XV_Alim_Douche(
    Enable := Option_Douche AND NOT Option_Debitmetre_Douche,
    Type_Consigne := FALSE,
    Mode_Vidange := FALSE,
    Cons_Pos_Dem := 0.0,
    Cmd_Ouv_Dem := Cmd_Appli_Vanne_Alim_Douche,
    Info_Mes_Pos := 0.0,
    Presence_Fdc := 3,
    Info_Fdc_Ouvert := E_Vanne_Alim_Douche_Ouv,
    Info_Fdc_Ferme := E_Vanne_Alim_Douche_Ferm,
    Secu_Niveau_Haut := Defaut_Debordement_Douche,
    Defaut_Alim_Eau := Defaut_General_Alim_Eau,
    Control_Discrodance := TRUE,
    Hyst_Al_Discord := 0.0,
    Tempo_Discord_TOR := T#15s,
    EF_Forcage := EF_Cmd_Vanne_Alim_Douche,
    F_STOR_Registre := F_Cmd_Vanne_Alim_Douche,
    F_SAN_Registre := 0.0,
    In_SCL_MIN_REAL := 0.0,
    In_SCL_OUT_REAL := 100.0,
    SAN_MIN := 0.0,
    SAN_MAX := 32767.0); // Registre_V1
S_Cmd_Vanne_Alim_Douche := XV_Alim_Douche.STOR_Cmd_Ouv_Registre;
Defaut_Discord_Vanne_Alim_Douche_Ouv := XV_Alim_Douche.Def_Discordance_Ouverture;
Defaut_Discord_Vanne_Alim_Douche_Ferm := XV_Alim_Douche.Def_Discordance_Fermeture;
XV_Alim_Douchette(
    Enable := Option_Douchette,
    Type_Consigne := FALSE,
    Mode_Vidange := FALSE,
    Cons_Pos_Dem := 0.0,
    Cmd_Ouv_Dem := Cmd_Appli_Vanne_Alim_Douchette,
    Info_Mes_Pos := 0.0,
    Presence_Fdc := 3,
    Info_Fdc_Ouvert := E_Vanne_Alim_Douchette_Ouv,
    Info_Fdc_Ferme := E_Vanne_Alim_Douchette_Ferm,
    Secu_Niveau_Haut := Defaut_Debordement_Douche,
    Defaut_Alim_Eau := Defaut_General_Alim_Eau,
    Control_Discrodance := TRUE,
    Hyst_Al_Discord := 0.0,
    Tempo_Discord_TOR := T#15s,
    EF_Forcage := EF_Cmd_Vanne_Alim_Douchette,
    F_STOR_Registre := F_Cmd_Vanne_Alim_Douchette,
    F_SAN_Registre := 0.0,
    In_SCL_MIN_REAL := 0.0,
    In_SCL_OUT_REAL := 100.0,
    SAN_MIN := 0.0,
    SAN_MAX := 32767.0); // Registre_V1
S_Cmd_Vanne_Alim_Douchette := XV_Alim_Douchette.STOR_Cmd_Ouv_Registre;
Defaut_Discord_Vanne_Alim_Douchette_Ouv := XV_Alim_Douchette.Def_Discordance_Ouverture;
Defaut_Discord_Vanne_Alim_Douchette_Ferm := XV_Alim_Douchette.Def_Discordance_Fermeture;
XV_Alim_Lavabo(
    Enable := Option_Lavabo AND NOT Option_Debitmetre_Lavabo,
    Type_Consigne := FALSE,
    Mode_Vidange := FALSE,
    Cons_Pos_Dem := 0.0,
    Cmd_Ouv_Dem := Cmd_Appli_Vanne_Alim_Lavabo,
    Info_Mes_Pos := 0.0,
    Presence_Fdc := 3,
    Info_Fdc_Ouvert := E_Vanne_Alim_Lavabo_Ouv,
    Info_Fdc_Ferme := E_Vanne_Alim_Lavabo_Ferm,
    Secu_Niveau_Haut := Defaut_Debordement_Lavabo,
    Defaut_Alim_Eau := Defaut_General_Alim_Eau,
    Control_Discrodance := TRUE,
    Hyst_Al_Discord := 0.0,
    Tempo_Discord_TOR := T#15s,
    EF_Forcage := EF_Cmd_Vanne_Alim_Lavabo,
    F_STOR_Registre := F_Cmd_Vanne_Alim_Lavabo,
    F_SAN_Registre := 0.0,
    In_SCL_MIN_REAL := 0.0,
    In_SCL_OUT_REAL := 100.0,
    SAN_MIN := 0.0,
    SAN_MAX := 32767.0); // Registre_V1
S_Cmd_Vanne_Alim_Lavabo := XV_Alim_Lavabo.STOR_Cmd_Ouv_Registre;
Defaut_Discord_Vanne_Alim_Lavabo_Ouv := XV_Alim_Lavabo.Def_Discordance_Ouverture;
Defaut_Discord_Vanne_Alim_Lavabo_Ferm := XV_Alim_Lavabo.Def_Discordance_Fermeture;
XV_Vid_Douche(
    Enable := Option_Douche,
    Type_Consigne := FALSE,
    Mode_Vidange := TRUE,
    Cons_Pos_Dem := 0.0,
    Cmd_Ouv_Dem := Cmd_Appli_Vanne_Vid_Douche OR Mode_Cabine_Libre,
    Info_Mes_Pos := 0.0,
    Presence_Fdc := 3,
    Info_Fdc_Ouvert := E_Vanne_Vidange_Douche_Ouv,
    Info_Fdc_Ferme := E_Vanne_Vidange_Douche_Ferm,
    Secu_Niveau_Haut := Defaut_Debordement_Douche,
    Defaut_Alim_Eau := FALSE,
    Control_Discrodance := TRUE,
    Hyst_Al_Discord := 0.0,
    Tempo_Discord_TOR := T#15s,
    EF_Forcage := EF_Cmd_Vanne_Vid_Douche,
    F_STOR_Registre := F_Cmd_Vanne_Vid_Douche,
    F_SAN_Registre := 0.0,
    In_SCL_MIN_REAL := 0.0,
    In_SCL_OUT_REAL := 100.0,
    SAN_MIN := 0.0,
    SAN_MAX := 32767.0); // Registre_V1
S_Cmd_Vanne_Vid_Douche := XV_Vid_Douche.STOR_Cmd_Ouv_Registre;
Defaut_Discord_Vanne_Vid_Douche_Ouv := XV_Vid_Douche.Def_Discordance_Ouverture;
Defaut_Discord_Vanne_Vid_Douche_Ferm := XV_Vid_Douche.Def_Discordance_Fermeture;
XV_Vid_Lavabo(
    Enable := Option_Lavabo,
    Type_Consigne := FALSE,
    Mode_Vidange := TRUE,
    Cons_Pos_Dem := 0.0,
    Cmd_Ouv_Dem := Cmd_Appli_Vanne_Vid_Lavabo OR Mode_Cabine_Libre,
    Info_Mes_Pos := 0.0,
    Presence_Fdc := 3,
    Info_Fdc_Ouvert := E_Vanne_Vidange_Lavabo_Ouv,
    Info_Fdc_Ferme := E_Vanne_Vidange_Lavabo_Ferm,
    Secu_Niveau_Haut := Defaut_Debordement_Lavabo,
    Defaut_Alim_Eau := FALSE,
    Control_Discrodance := TRUE,
    Hyst_Al_Discord := 0.0,
    Tempo_Discord_TOR := T#15s,
    EF_Forcage := EF_Cmd_Vanne_Vid_Lavabo,
    F_STOR_Registre := F_Cmd_Vanne_Vid_Lavabo,
    F_SAN_Registre := 0.0,
    In_SCL_MIN_REAL := 0.0,
    In_SCL_OUT_REAL := 100.0,
    SAN_MIN := 0.0,
    SAN_MAX := 32767.0); // Registre_V1
S_Cmd_Vanne_Vid_Lavabo := XV_Vid_Lavabo.STOR_Cmd_Ouv_Registre;
Defaut_Discord_Vanne_Vid_Lavabo_Ouv := XV_Vid_Lavabo.Def_Discordance_Ouverture;
Defaut_Discord_Vanne_Vid_Lavabo_Ferm := XV_Vid_Lavabo.Def_Discordance_Fermeture;
XV_Electrovanne_Douche(
    Enable := Option_Debitmetre_Douche,
    Type_Consigne := FALSE,
    Mode_Vidange := FALSE,
    Cons_Pos_Dem := 0.0,
    Cmd_Ouv_Dem := Cmd_Appli_ElectroValve_Alim_Douche,
    Info_Mes_Pos := 0.0,
    Presence_Fdc := 0,
    Info_Fdc_Ouvert := FALSE,
    Info_Fdc_Ferme := FALSE,
    Secu_Niveau_Haut := Defaut_Debordement_Douche,
    Defaut_Alim_Eau := Defaut_General_Alim_Eau,
    Control_Discrodance := TRUE,
    Hyst_Al_Discord := 0.0,
    Tempo_Discord_TOR := T#15s,
    EF_Forcage := EF_Cmd_ElectroValve_Alim_Douche,
    F_STOR_Registre := F_Cmd_ElectroValve_Alim_Douche,
    F_SAN_Registre := 0.0,
    In_SCL_MIN_REAL := 0.0,
    In_SCL_OUT_REAL := 100.0,
    SAN_MIN := 0.0,
    SAN_MAX := 32767.0); // Registre_V1
S_Cmd_ElectroValve_Alim_Douche := XV_Electrovanne_Douche.STOR_Cmd_Ouv_Registre;
XV_Electrovanne_Lavabo(
    Enable := Option_Debitmetre_Lavabo,
    Type_Consigne := FALSE,
    Mode_Vidange := FALSE,
    Cons_Pos_Dem := 0.0,
    Cmd_Ouv_Dem := Cmd_Appli_ElectroValve_Alim_Lavabo,
    Info_Mes_Pos := 0.0,
    Presence_Fdc := 0,
    Info_Fdc_Ouvert := FALSE,
    Info_Fdc_Ferme := FALSE,
    Secu_Niveau_Haut := Defaut_Debordement_Lavabo,
    Defaut_Alim_Eau := Defaut_General_Alim_Eau,
    Control_Discrodance := TRUE,
    Hyst_Al_Discord := 0.0,
    Tempo_Discord_TOR := T#15s,
    EF_Forcage := EF_Cmd_ElectroValve_Alim_Lavabo,
    F_STOR_Registre := F_Cmd_ElectroValve_Alim_Lavabo,
    F_SAN_Registre := 0.0,
    In_SCL_MIN_REAL := 0.0,
    In_SCL_OUT_REAL := 100.0,
    SAN_MIN := 0.0,
    SAN_MAX := 32767.0); // Registre_V1
S_Cmd_ElectroValve_Alim_Lavabo := XV_Electrovanne_Lavabo.STOR_Cmd_Ouv_Registre;
Prise_Cabine(
    Enable := Option_Prise,
    Cmd_Prise := SEL(EF_Cmd_PC_Cab, TRUE, F_Cmd_PC_Cab),
    Cabine_Seche := Option_Cabine_Seche,
    Statut_Ferm_Reg_Douche := TRUE,
    Statut_Ferm_Lavabo := TRUE,
    Statut_Electrovanne_Douche := FALSE,
    Statut_Electrovanne_Lavabo := FALSE,
    Statut_Def_Prise_Porte_Ouverte := Def_Prise_Porte_Ouverte,
    Statut_Def_Discord_Alim_Prise := Def_Discord_Alim_Prise,
    Statut_Defaut_Discord_PC_Cab := Defaut_Discord_PC_Cab); // Prise
S_Cmd_PC_Cab := Prise_Cabine.STOR_Prise;
XV_Vanne_Souf_Bas_Deb(
    Enable := Option_Bas_Debit,
    Type_Consigne := FALSE,
    Mode_Vidange := FALSE,
    Cons_Pos_Dem := 0.0,
    Cmd_Ouv_Dem := Cmd_Appli_Vanne_Souf_Bas_Deb,
    Info_Mes_Pos := 0.0,
    Presence_Fdc := 3,
    Info_Fdc_Ouvert := E_Vanne_Souf_Bas_Deb_Ouv,
    Info_Fdc_Ferme := E_Vanne_Souf_Bas_Deb_Ferm,
    Secu_Niveau_Haut := FALSE,
    Defaut_Alim_Eau := FALSE,
    Control_Discrodance := TRUE,
    Hyst_Al_Discord := 0.0,
    Tempo_Discord_TOR := T#95s,
    EF_Forcage := EF_Vanne_Souf_Bas_Deb,
    F_STOR_Registre := F_Vanne_Souf_Bas_Deb,
    F_SAN_Registre := 0.0,
    In_SCL_MIN_REAL := 0.0,
    In_SCL_OUT_REAL := 100.0,
    SAN_MIN := 0.0,
    SAN_MAX := 32767.0); // Registre_V1
S_Cmd_Vanne_Souf_Bas_Deb := XV_Vanne_Souf_Bas_Deb.STOR_Cmd_Ouv_Registre;
Defaut_Discord_Vanne_Souf_Bas_Deb_Ouv := XV_Vanne_Souf_Bas_Deb.Def_Discordance_Ouverture;
Defaut_Discord_Vanne_Souf_Bas_Deb_Ferm := XV_Vanne_Souf_Bas_Deb.Def_Discordance_Fermeture;
XV_Vanne_Ext_Bas_Deb(
    Enable := Option_Bas_Debit,
    Type_Consigne := FALSE,
    Mode_Vidange := FALSE,
    Cons_Pos_Dem := 0.0,
    Cmd_Ouv_Dem := Cmd_Appli_Vanne_Ext_Bas_Deb,
    Info_Mes_Pos := 0.0,
    Presence_Fdc := 3,
    Info_Fdc_Ouvert := E_Vanne_Ext_Bas_Deb_Ouv,
    Info_Fdc_Ferme := E_Vanne_Ext_Bas_Deb_Ferm,
    Secu_Niveau_Haut := FALSE,
    Defaut_Alim_Eau := FALSE,
    Control_Discrodance := TRUE,
    Hyst_Al_Discord := 0.0,
    Tempo_Discord_TOR := T#95s,
    EF_Forcage := EF_Vanne_Ext_Bas_Deb,
    F_STOR_Registre := F_Vanne_Ext_Bas_Deb,
    F_SAN_Registre := 0.0,
    In_SCL_MIN_REAL := 0.0,
    In_SCL_OUT_REAL := 100.0,
    SAN_MIN := 0.0,
    SAN_MAX := 32767.0); // Registre_V1
S_Cmd_Vanne_Ext_Bas_Deb := XV_Vanne_Ext_Bas_Deb.STOR_Cmd_Ouv_Registre;
Defaut_Discord_Vanne_Ext_Bas_Deb_Ouv := XV_Vanne_Ext_Bas_Deb.Def_Discordance_Ouverture;
Defaut_Discord_Vanne_Ext_Bas_Deb_Ferm := XV_Vanne_Ext_Bas_Deb.Def_Discordance_Fermeture;
Reg_Etanche_Souf(
    Enable := Option_Reg_Etanche_Souf,
    Type_Consigne := FALSE,
    Mode_Vidange := FALSE,
    Cons_Pos_Dem := 0.0,
    Cmd_Ouv_Dem := Cmd_Appli_Reg_Etanche_Souf,
    Info_Mes_Pos := 0.0,
    Presence_Fdc := 0,
    Info_Fdc_Ouvert := FALSE,
    Info_Fdc_Ferme := FALSE,
    Secu_Niveau_Haut := FALSE,
    Defaut_Alim_Eau := FALSE,
    Control_Discrodance := FALSE,
    Hyst_Al_Discord := 0.0,
    Tempo_Discord_TOR := T#40s,
    EF_Forcage := EF_Cmd_Reg_Etanche_Souf,
    F_STOR_Registre := F_Cmd_Reg_Etanche_Souf,
    F_SAN_Registre := 0.0,
    In_SCL_MIN_REAL := 0.0,
    In_SCL_OUT_REAL := 100.0,
    SAN_MIN := 0.0,
    SAN_MAX := 32767.0); // Registre_V1
S_Cmd_Reg_Etanche_Souf := Reg_Etanche_Souf.STOR_Cmd_Ouv_Registre;
XV_Alim_NEP(
    Enable := Option_NEP,
    Type_Consigne := FALSE,
    Mode_Vidange := FALSE,
    Cons_Pos_Dem := 0.0,
    Cmd_Ouv_Dem := Cmd_Appli_Vanne_Alim_NEP,
    Info_Mes_Pos := 0.0,
    Presence_Fdc := 3,
    Info_Fdc_Ouvert := E_Vanne_Alim_NEP_Ouv,
    Info_Fdc_Ferme := E_Vanne_Alim_NEP_Ferm,
    Secu_Niveau_Haut := FALSE,
    Defaut_Alim_Eau := FALSE,
    Control_Discrodance := TRUE,
    Hyst_Al_Discord := 0.0,
    Tempo_Discord_TOR := T#95s,
    EF_Forcage := EF_Vanne_Alim_NEP,
    F_STOR_Registre := F_Vanne_Alim_NEP,
    F_SAN_Registre := 0.0,
    In_SCL_MIN_REAL := 0.0,
    In_SCL_OUT_REAL := 100.0,
    SAN_MIN := 0.0,
    SAN_MAX := 32767.0); // Registre_V1
S_Cmd_Vanne_NEP := XV_Alim_NEP.STOR_Cmd_Ouv_Registre;
Defaut_Discord_Vanne_Alim_NEP_Ouv := XV_Alim_NEP.Def_Discordance_Ouverture;
Defaut_Discord_Vanne_Alim_NEP_Ferm := XV_Alim_NEP.Def_Discordance_Fermeture;
Y_Verin_WC_GV(
    Enable := Option_WC_GV,
    Type_Consigne := FALSE,
    Mode_Vidange := FALSE,
    Cons_Pos_Dem := 0.0,
    Cmd_Ouv_Dem := Cmd_Appli_Verin_WC_GV,
    Info_Mes_Pos := 0.0,
    Presence_Fdc := 0,
    Info_Fdc_Ouvert := FALSE,
    Info_Fdc_Ferme := FALSE,
    Secu_Niveau_Haut := FALSE,
    Defaut_Alim_Eau := FALSE,
    Control_Discrodance := FALSE,
    Hyst_Al_Discord := 0.0,
    Tempo_Discord_TOR := T#95s,
    EF_Forcage := EF_Cmd_Verin_WC_GV,
    F_STOR_Registre := F_Cmd_Verin_WC_GV,
    F_SAN_Registre := 0.0,
    In_SCL_MIN_REAL := 0.0,
    In_SCL_OUT_REAL := 100.0,
    SAN_MIN := 0.0,
    SAN_MAX := 32767.0); // Registre_V1
S_Cmd_Appli_Verin_WC_GV := Y_Verin_WC_GV.STOR_Cmd_Ouv_Registre;
Y_Verin_WC_PV(
    Enable := Option_WC_PV,
    Type_Consigne := FALSE,
    Mode_Vidange := FALSE,
    Cons_Pos_Dem := 0.0,
    Cmd_Ouv_Dem := Cmd_Appli_Verin_WC_PV,
    Info_Mes_Pos := 0.0,
    Presence_Fdc := 0,
    Info_Fdc_Ouvert := FALSE,
    Info_Fdc_Ferme := FALSE,
    Secu_Niveau_Haut := FALSE,
    Defaut_Alim_Eau := FALSE,
    Control_Discrodance := FALSE,
    Hyst_Al_Discord := 0.0,
    Tempo_Discord_TOR := T#95s,
    EF_Forcage := EF_Cmd_Verin_WC_PV,
    F_STOR_Registre := F_Cmd_Verin_WC_PV,
    F_SAN_Registre := 0.0,
    In_SCL_MIN_REAL := 0.0,
    In_SCL_OUT_REAL := 100.0,
    SAN_MIN := 0.0,
    SAN_MAX := 32767.0); // Registre_V1
S_Cmd_Appli_Verin_WC_PV := Y_Verin_WC_PV.STOR_Cmd_Ouv_Registre;
Gestion_EA_WC(
    OUTPUT_1 := Y_Verin_WC_GV.STOR_Cmd_Ouv_Registre,
    OUTPUT_2 := Y_Verin_WC_PV.STOR_Cmd_Ouv_Registre,
    OUTPUT_3 := FALSE,
    OUTPUT_4 := FALSE,
    SWITCH_SEQUENCE := 0); // Sontay_4RM
S_Cons_Module_Sontay := Gestion_EA_WC.OUT_SAN;

END_PROGRAM

// ---- POUs/Block/Autres/Sontay_4RM.TcPOU
FUNCTION_BLOCK Sontay_4RM
VAR_INPUT
	OUTPUT_1 :BOOL;
	OUTPUT_2 :BOOL;
	OUTPUT_3 :BOOL;
	OUTPUT_4 :BOOL;
	SWITCH_SEQUENCE :INT; (*0=Sequenced / 1=Staged / 1=Binary*)
END_VAR
VAR_OUTPUT
	OUT_SAN :INT;
END_VAR
VAR
	Sortie_Calcul_Sequenced :INT;
	SCL_Sequenced: SCL;
END_VAR

(*Bloc de fonction permettant de gérer le module IO-RM4 de sontay*)

(*Version Sequenced*)
IF (SWITCH_SEQUENCE = 0)
	THEN
	IF (OUTPUT_1) (*La valeur doit être comprise entre 2 et 4 VDC*)
		THEN
		Sortie_Calcul_Sequenced := 3;
	END_IF;
	IF (OUTPUT_2) (*La valeur doit être comprise entre 4 et 6 VDC*)
		THEN
		Sortie_Calcul_Sequenced := 5;
	END_IF;
	IF (OUTPUT_3) (*La valeur doit être comprise entre 6 et 8 VDC*)
		THEN
		Sortie_Calcul_Sequenced := 7;
	END_IF;
	IF (OUTPUT_4) (*La valeur doit être comprise entre 8 et 10 VDC*)
		THEN
		Sortie_Calcul_Sequenced := 9;
	END_IF;
	IF (NOT OUTPUT_1 AND NOT OUTPUT_2 AND NOT OUTPUT_3 AND NOT OUTPUT_4)
		THEN
		Sortie_Calcul_Sequenced := 0;
	END_IF;
END_IF;

(*Mise à l'échelle de la valeur*)
SCL_Sequenced(
	IN_INT:= Sortie_Calcul_Sequenced,
	LIM_MIN_IN_REAL:= 0,
	LIM_MAX_IN_REAL:= 10,
	LIM_MIN_OUT_REAL:= 0.0,
	LIM_MAX_OUT_REAL:= 32767.0,
	OUT_INT=> OUT_SAN);

END_FUNCTION_BLOCK

// ---- POUs/s_InterCom_Esclave.TcPOU
PROGRAM s_InterCom_Esclave
VAR
	fbServer						: FB_LocalServer;
	bEnableServer				: BOOL := TRUE;
	fbSocketCloseAll				: FB_SocketCloseAll :=  ( sSrvNetID := '', tTimeout := DEFAULT_ADS_TIMEOUT );
	bCloseAll					: BOOL := TRUE;
	TON_Def_Client: TON;
	TON_Def_Com: TON;
	i :INT;
END_VAR

fbServer(  sLocalHost := Own_Ip_Adress, nLocalPort := 200 );

IF (bCloseAll OR NOT Option_InterCom) THEN (*On PLC reset or program download close all old connections *)
	bCloseAll := FALSE;
	fbSocketCloseAll( bExecute:= TRUE );
ELSE
	fbSocketCloseAll( bExecute:= FALSE );
END_IF

IF (Option_InterCom)
	THEN
	IF NOT fbSocketCloseAll.bBusy THEN
		fbServer( bEnable := bEnableServer );
	END_IF
	(*Gestion du defaut de communication*)
	TON_Def_Client(IN:= (fbServer.nAcceptedClients = 0), PT:= T#10s); (*Si aucun accepté au démarrage de l'automate*)
	TON_Def_Com(IN:= (fbServer.fbRemoteClient[1].fbServerDataExcha.bError OR TON_Def_Client.Q), PT:= T#20s);
	Defaut_Com_Client := TON_Def_Com.Q;
	(*Initilisation des lectures et ecritures en cas de défaut com*)
	IF (Defaut_Com_Client)
		THEN
		FOR i := 0 TO 29 BY 1 DO
		Tab_Com_Send[i] := 0;
		Tab_Com_Receive[i] := 0;
		END_FOR;
	END_IF;
	ELSE
	TON_Def_Client(IN:=FALSE);
	Defaut_Com_Client := FALSE;
	FOR i := 0 TO 29 BY 1 DO
	Tab_Com_Send[i] := 0;
	Tab_Com_Receive[i] := 0;
	END_FOR;
END_IF;

END_PROGRAM

// ---- POUs/Block/Com_Ip/FB_LocalServer.TcPOU
FUNCTION_BLOCK FB_LocalServer
VAR_INPUT
	sLocalHost					: STRING(15);(* own IP address! *)
	nLocalPort					: UDINT := 0;
	bEnable						: BOOL;
END_VAR
VAR_OUTPUT
	bListening					: BOOL;
	hListener 					: T_HSOCKET;
	nAcceptedClients				: UDINT;
	bBusy						: BOOL;
	bError 						: BOOL;
	nErrId						: UDINT;
END_VAR
VAR
	fbListen	 					: FB_SocketListen := ( sSrvNetID := '', tTimeout := DEFAULT_ADS_TIMEOUT );
	fbClose						: FB_SocketClose := ( sSrvNetID := '', tTimeout := DEFAULT_ADS_TIMEOUT );
	fbConnectTON				: TON := ( PT := T#3s );
	eStep						: E_ServerSteps;
	fbRemoteClient				: ARRAY[1..1] OF FB_RemoteClient;
	i							: UDINT;
END_VAR

CASE eStep OF

	SERVER_STATE_IDLE:
		IF bEnable XOR bListening THEN
			bBusy := TRUE;
			bError := FALSE;
			nErrId := 0;
			IF bEnable THEN
				fbConnectTON( IN := FALSE );
				eStep := SERVER_STATE_LISTENER_OPEN_START;
			ELSE
				eStep := SERVER_STATE_REMOTE_CLIENTS_CLOSE;
			END_IF
		ELSIF bListening THEN
			eStep := SERVER_STATE_REMOTE_CLIENTS_COMM;
		END_IF

	SERVER_STATE_LISTENER_OPEN_START:
		fbConnectTON( IN := TRUE, PT := PLCPRJ_RECONNECT_TIME );
		IF fbConnectTON.Q THEN
			fbConnectTON( IN := FALSE );
			fbListen(  bExecute := FALSE  );
			fbListen(	sLocalHost	:= sLocalHost,
					nLocalPort	:= nLocalPort,
					bExecute	:= TRUE );
			eStep := SERVER_STATE_LISTENER_OPEN_WAIT;
		END_IF

	SERVER_STATE_LISTENER_OPEN_WAIT:
		fbListen( bExecute := FALSE );
		IF NOT fbListen.bBusy THEN
			IF NOT fbListen.bError THEN
				bListening 	:= TRUE;
				hListener 	:= fbListen.hListener;
				eStep 		:= SERVER_STATE_IDLE;
				LogMessage( 'LISTENER socket OPENED!', hListener );
			ELSE
				LogError( 'FB_SocketListen',  fbListen.nErrId );
				nErrId := fbListen.nErrId;
				eStep := SERVER_STATE_ERROR;
			END_IF
		END_IF

	SERVER_STATE_REMOTE_CLIENTS_COMM:
		eStep := SERVER_STATE_IDLE;
		nAcceptedClients := 0;

		FOR i:= 1 TO MAX_CLIENT_CONNECTIONS DO
			fbRemoteClient[ i ]( hListener := hListener, bEnable := TRUE );
			IF NOT  fbRemoteClient[ i ].bBusy AND fbRemoteClient[ i ].bError THEN (*FB_SocketAccept returned error!*)
				eStep := SERVER_STATE_REMOTE_CLIENTS_CLOSE;
				EXIT;
			END_IF

			(* count the number of connected remote clients *)
			IF fbRemoteClient[ i ].bAccepted THEN
				nAcceptedClients := nAcceptedClients + 1;
			END_IF

		END_FOR

	SERVER_STATE_REMOTE_CLIENTS_CLOSE:
		nAcceptedClients := 0;
		eStep := SERVER_STATE_LISTENER_CLOSE_START; (* close listener socket too *)
		FOR i:= 1 TO MAX_CLIENT_CONNECTIONS DO
			fbRemoteClient[ i ]( bEnable := FALSE );(* close all remote client (accepted) sockets *)
			(* check if all remote client sockets are closed *)
			IF fbRemoteClient[ i ].bAccepted THEN
				eStep := SERVER_STATE_REMOTE_CLIENTS_CLOSE; (* stay here and close all remote clients first *)
				nAcceptedClients := nAcceptedClients + 1;
			END_IF
		END_FOR

	SERVER_STATE_LISTENER_CLOSE_START:
		fbClose( bExecute := FALSE );
		fbClose(	hSocket	:= hListener,
				bExecute:= TRUE );
		eStep := SERVER_STATE_LISTENER_CLOSE_WAIT;

	SERVER_STATE_LISTENER_CLOSE_WAIT:
		fbClose( bExecute := FALSE );
		IF NOT fbClose.bBusy THEN
			LogMessage( 'LISTENER socket CLOSED!', hListener );
			bListening := FALSE;
			MEMSET( ADR(hListener), 0, SIZEOF(hListener));
			IF fbClose.bError THEN
				LogError( 'FB_SocketClose (listener)',  fbClose.nErrId );
				nErrId := fbClose.nErrId;
				eStep := SERVER_STATE_ERROR;
			ELSE
				bBusy := FALSE;
				bError := FALSE;
				nErrId := 0;
				eStep := SERVER_STATE_IDLE;
			END_IF
		END_IF

	SERVER_STATE_ERROR:
		bError := TRUE;
		IF bListening THEN
			eStep := SERVER_STATE_REMOTE_CLIENTS_CLOSE;
		ELSE
			bBusy := FALSE;
			eStep := SERVER_STATE_IDLE;
		END_IF

END_CASE

END_FUNCTION_BLOCK

// ---- POUs/Block/Com_Ip/FB_RemoteClient.TcPOU
FUNCTION_BLOCK FB_RemoteClient
VAR_INPUT
	hListener				: T_HSOCKET;
	bEnable 				: BOOL;
END_VAR
VAR_OUTPUT
	bAccepted			: BOOL;
	hSocket				: T_HSOCKET;
	bBusy				: BOOL;
	bError 				: BOOL;
	nErrID				: UDINT;
	sFromClient			: T_MaxString;
END_VAR
VAR
	fbAccept 			: FB_SocketAccept := ( sSrvNetID := '', tTimeout := DEFAULT_ADS_TIMEOUT );
	fbClose				: FB_SocketClose := ( sSrvNetID := '', tTimeout := DEFAULT_ADS_TIMEOUT );
	fbServerDataExcha	: FB_ServerDataExcha;
	fbAcceptTON			: TON := ( PT := T#1s);
	eStep				: E_ClientSteps;
	R_TRIG_1: R_TRIG;
END_VAR

CASE eStep OF

	CLIENT_STATE_IDLE:
		IF bEnable XOR bAccepted THEN
			bBusy := TRUE;
			bError := FALSE;
			nErrId := 0;
			sFromClient := '';
			IF bEnable THEN
				fbAcceptTON( IN := FALSE );
				eStep := CLIENT_STATE_CONNECT_START;
			ELSE
				eStep := CLIENT_STATE_CLOSE_START;
			END_IF
		ELSIF bAccepted THEN
			eStep := CLIENT_STATE_DATAEXCHA_START;
		ELSE
			bBusy := FALSE;
		END_IF

	CLIENT_STATE_CONNECT_START:
		fbAcceptTON( IN := TRUE, PT := PLCPRJ_ACCEPT_POLLING_TIME );
		IF fbAcceptTON.Q THEN
			fbAcceptTON( IN := FALSE );
			fbAccept(  bExecute := FALSE  );
			fbAccept(	hListener := hListener,
						bExecute:= TRUE );
			eStep := CLIENT_STATE_CONNECT_WAIT;
		END_IF

	CLIENT_STATE_CONNECT_WAIT:
		fbAccept( bExecute := FALSE );
		IF NOT fbAccept.bBusy THEN
			IF NOT fbAccept.bError THEN
				IF fbAccept.bAccepted THEN
					bAccepted := TRUE;
					hSocket := fbAccept.hSocket;
					LogMessage( 'REMOTE client ACCEPTED!', hSocket );
				END_IF
				eStep := CLIENT_STATE_IDLE;
			ELSE
				LogError( 'FB_SocketAccept',  fbAccept.nErrId );
				nErrId := fbAccept.nErrId;
				eStep := CLIENT_STATE_ERROR;
			END_IF
		END_IF

	CLIENT_STATE_DATAEXCHA_START:
		fbServerDataExcha( bExecute := FALSE );
		fbServerDataExcha( 	hSocket := hSocket,
								bExecute := TRUE );
		eStep := CLIENT_STATE_DATAEXCHA_WAIT;

	CLIENT_STATE_DATAEXCHA_WAIT:
		fbServerDataExcha( bExecute := FALSE, sFromClient=>sFromClient );
		IF NOT fbServerDataExcha.bBusy THEN
			IF NOT fbServerDataExcha.bError THEN
				eStep := CLIENT_STATE_IDLE;
			ELSE
				(* possible errors are logged inside of fbServerDataExcha function block *)
				nErrId := fbServerDataExcha.nErrID;
				eStep := CLIENT_STATE_ERROR;
			END_IF
		END_IF

	CLIENT_STATE_CLOSE_START:
		fbClose( bExecute := FALSE );
		fbClose(	hSocket:= hSocket,
				bExecute:= TRUE );
		eStep := CLIENT_STATE_CLOSE_WAIT;

	CLIENT_STATE_CLOSE_WAIT:
		fbClose( bExecute := FALSE );
		IF NOT fbClose.bBusy THEN
			LogMessage( 'REMOTE client CLOSED!', hSocket );
			bAccepted := FALSE;
			MEMSET( ADR( hSocket ), 0, SIZEOF( hSocket ) );
			IF fbClose.bError THEN
				LogError( 'FB_SocketClose (remote client)', fbClose.nErrId );
				nErrId := fbClose.nErrId;
				eStep := CLIENT_STATE_ERROR;
			ELSE
				bBusy := FALSE;
				bError := FALSE;
				nErrId := 0;
				eStep := CLIENT_STATE_IDLE;
			END_IF
		END_IF

	CLIENT_STATE_ERROR:
		bError := TRUE;
		IF bAccepted THEN
			eStep := CLIENT_STATE_CLOSE_START;
		ELSE
			eStep := CLIENT_STATE_IDLE;
			bBusy := FALSE;
		END_IF
END_CASE

R_TRIG_1(CLK:= fbServerDataExcha.bError);
IF(R_TRIG_1.Q)
	THEN
	eStep := CLIENT_STATE_ERROR;
END_IF;

END_FUNCTION_BLOCK

// ---- POUs/Block/Com_Ip/FB_ServerDataExcha.TcPOU
FUNCTION_BLOCK FB_ServerDataExcha
VAR_INPUT
	hSocket			: T_HSOCKET;
	bExecute		: BOOL;
END_VAR
VAR_OUTPUT
	bBusy			: BOOL;
	bError 			: BOOL;
	nErrID			: UDINT;
	sFromClient		: T_MaxString;
END_VAR
VAR
	fbSocketReceive	: FB_SocketReceive := ( sSrvNetId := '', tTimeout := DEFAULT_ADS_TIMEOUT );
	fbSocketSend	: FB_SocketSend :=  ( sSrvNetId := '', tTimeout := DEFAULT_ADS_TIMEOUT );
	eStep			: E_DataExchaSteps;
	RisingEdge		: R_TRIG;
	fbReceiveTON	: TON;
	fbDisconnectTON 	: TON;
	cbReceived, startPos, endPos, idx	: UDINT;
	cbFrame			: UDINT;
	rxBuffer			: ARRAY[0..1000] OF BYTE;
END_VAR

RisingEdge( CLK := bExecute );
CASE eStep OF

	DATAEXCHA_STATE_IDLE:
		IF RisingEdge.Q THEN
			bBusy 	:= TRUE;
			bError 	:= FALSE;
			nErrId 	:= 0;
			fbDisconnectTON( IN := FALSE, PT := T#0s );(* disable timeout check first *)
			fbReceiveTON( IN := FALSE, PT := T#0s ); (* receive first request immediately *)
			eStep 	:= DATAEXCHA_STATE_RECEIVE_START;
		END_IF

	DATAEXCHA_STATE_RECEIVE_START: (* Receive remote client data *)
		fbReceiveTON(  IN := TRUE );
		IF fbReceiveTON.Q THEN
			fbReceiveTON( IN := FALSE );
			fbSocketReceive( bExecute := FALSE );
			fbSocketReceive( 	hSocket		:= hSocket,
							pDest		:= ADR( Tab_Com_Receive ),			(*ADR( rxBuffer ) + cbReceived,*)
							cbLen		:= SIZEOF( Tab_Com_Receive ),		(*SIZEOF( rxBuffer ) - cbReceived,*)
							bExecute	:= TRUE );
			eStep := DATAEXCHA_STATE_RECEIVE_WAIT;
		END_IF

	DATAEXCHA_STATE_RECEIVE_WAIT:
		fbSocketReceive( bExecute := FALSE );
		IF NOT fbSocketReceive.bBusy THEN
			IF NOT fbSocketReceive.bError THEN

				IF (fbSocketReceive.nRecBytes > 0) THEN(* bytes received *)

					startPos 		:= cbReceived;(* rxBuffer array index of first data byte *)
					endPos  		:= cbReceived + fbSocketReceive.nRecBytes  - 1;(* rxBuffer array index of last data byte *)
					cbReceived 	:= cbReceived + fbSocketReceive.nRecBytes;(* calculate the number of received data bytes *)
					cbFrame		:= 0;(* reset frame length *)

					IF cbReceived < SIZEOF( sFromClient ) THEN(* no overflow *)

						fbReceiveTON( IN := FALSE, PT := T#0s ); (* bytes received => increase the read (polling) speed *)
						fbDisconnectTON( IN := FALSE, PT := PLCPRJ_RECEIVE_TIMEOUT );(* bytes received => disable timeout check *)

						(* search for string end delimiter *)
						FOR idx := startPos TO endPos BY 1 DO
							IF rxBuffer[idx] = 0 THEN(* string end delimiter found *)
								cbFrame := idx + 1;(* calculate the length of the received string (inclusive the end delimiter) *)
								MEMCPY(  ADR( sFromClient ), ADR( rxBuffer ), cbFrame );(* copy the received string to the output variable (inclusive the end delimiter) *)
								MEMMOVE( ADR( rxBuffer ), ADR( rxBuffer[cbFrame] ),  cbReceived - cbFrame  );(* move the reamaining data bytes *)
								cbReceived := cbReceived - cbFrame;(* recalculate the reamaining data byte length *)
								eStep := DATAEXCHA_STATE_SEND_START;
								EXIT;
							END_IF
						END_FOR

					ELSE(* there is no more free read buffer space => the answer string should be terminated *)
						LogError( 'FB_SocketReceive (remote client)',  PLCPRJ_ERROR_RECEIVE_BUFFER_OVERFLOW );
						nErrId := PLCPRJ_ERROR_RECEIVE_BUFFER_OVERFLOW;(* buffer overflow !*)
						eStep := DATAEXCHA_STATE_ERROR;
					END_IF

				ELSE(* no bytes received *)
					fbReceiveTON( IN := FALSE, PT := PLCPRJ_RECEIVE_POLLING_TIME );(* no bytes received => decrease the read (polling) speed *)
					fbDisconnectTON( IN := TRUE, PT := PLCPRJ_RECEIVE_TIMEOUT );(* no bytes received => enable timeout check*)
					IF fbDisconnectTON.Q THEN (* timeout error*)
						fbDisconnectTON( IN := FALSE );
						LogError( 'FB_SocketReceive (remote client)',  PLCPRJ_ERROR_RECEIVE_TIMEOUT );
						nErrID := PLCPRJ_ERROR_RECEIVE_TIMEOUT;
						eStep := DATAEXCHA_STATE_ERROR;
					ELSE(* repeat reading *)
						eStep := DATAEXCHA_STATE_RECEIVE_START; (* repeat reading *)
					END_IF
				END_IF
			ELSE(* receive error *)
				LogError( 'FB_SocketReceive (remote client)',  fbSocketReceive.nErrId );
				nErrId := fbSocketReceive.nErrId;
				eStep := DATAEXCHA_STATE_ERROR;
			END_IF
		END_IF

	DATAEXCHA_STATE_SEND_START:
		fbSocketSend( bExecute := FALSE );
		fbSocketSend(	hSocket	:= hSocket,
						pSrc	:= ADR( Tab_Com_Send ),			(*ADR( sFromClient ),*)
						cbLen	:= SIZEOF( Tab_Com_Send ),		(*INT_TO_UDINT(LEN( sFromClient )) + 1,(* string length inclusive the zero delimiter *)*)
						bExecute:= TRUE );
		eStep := DATAEXCHA_STATE_SEND_WAIT;

	DATAEXCHA_STATE_SEND_WAIT:
		fbSocketSend( bExecute := FALSE );
		IF NOT fbSocketSend.bBusy THEN
			IF NOT fbSocketSend.bError THEN
				bBusy := FALSE;
				eStep := DATAEXCHA_STATE_IDLE;
			ELSE
				LogError( 'fbSocketSend (remote client)',  fbSocketSend.nErrId );
				nErrId := fbSocketSend.nErrId;
				eStep := DATAEXCHA_STATE_ERROR;
			END_IF
		END_IF

	DATAEXCHA_STATE_ERROR:
		bBusy := FALSE;
		bError := TRUE;
		cbReceived := 0;(* reset old received data bytes *)
		eStep := DATAEXCHA_STATE_IDLE;
END_CASE

END_FUNCTION_BLOCK

// ---- POUs/Block/Com_Ip/LogError.TcPOU
FUNCTION LogError : DINT
VAR_INPUT
	msg			: STRING;
	nErrId		: DWORD;
END_VAR
VAR
END_VAR

IF bLogDebugMessages THEN
	IF nErrId = 0 THEN
		LogError := ADSLOGSTR( ADSLOG_MSGTYPE_HINT OR ADSLOG_MSGTYPE_LOG, CONCAT( msg, '::No error!   %s'),'' );
	ELSIF ( nErrId AND 16#80000000) =16#80000000 THEN
		LogError := ADSLOGDINT( ADSLOG_MSGTYPE_ERROR OR ADSLOG_MSGTYPE_LOG, CONCAT( msg, ':: Win32 error: %d' ), DWORD_TO_DINT(SCODE_CODE( nErrId )) );
	ELSIF (nErrId AND 16#00008100) =16#00008100 THEN
		LogError := ADSLOGDINT( ADSLOG_MSGTYPE_ERROR OR ADSLOG_MSGTYPE_LOG, CONCAT( msg, '::Internal PLC sample project error: %d' ), DWORD_TO_DINT(nErrId) );
	ELSIF (nErrId AND 16#00008000) =16#00008000 THEN
		LogError := ADSLOGDINT( ADSLOG_MSGTYPE_ERROR OR ADSLOG_MSGTYPE_LOG, CONCAT( msg, '::Internal TCP/IP Connection Server error: %d' ), DWORD_TO_DINT(nErrId) );
	ELSE
		LogError := ADSLOGDINT( ADSLOG_MSGTYPE_ERROR OR ADSLOG_MSGTYPE_LOG, CONCAT( msg, '::TwinCAT System error: %d' ), DWORD_TO_DINT(nErrId) );
	END_IF
END_IF

END_FUNCTION

// ---- POUs/Block/Com_Ip/SCODE_CODE.TcPOU
FUNCTION SCODE_CODE : DWORD
VAR_INPUT
	sc		: DWORD;
END_VAR

SCODE_CODE := 16#FFFF AND sc;

END_FUNCTION

// ---- POUs/Block/Com_Ip/LogMessage.TcPOU
FUNCTION LogMessage : DINT
VAR_INPUT
	msg		: STRING;
	hSocket	: T_HSOCKET;
END_VAR
VAR
END_VAR

IF bLogDebugMessages THEN
	LogMessage := ADSLOGDINT( ADSLOG_MSGTYPE_HINT OR ADSLOG_MSGTYPE_LOG, CONCAT( msg, '::Internal handle: %d' ), UDINT_TO_DINT(hSocket.handle)  );
END_IF

END_FUNCTION

// ---- POUs/t_Enr_Variables.TcPOU
PROGRAM t_Enr_Variables
VAR
	WritePersistentData_1: WritePersistentData;
 	 bStart                : BOOL := TRUE;
  	 bError                : BOOL;
   	 bBusy                 : BOOL;
   	 nErrorId              : UDINT;
	Enregistrement_Manu: BOOL;
	TP_RAZ_Enr_Manu :TP;
END_VAR

TP_RAZ_Enr_Manu(IN:= Enregistrement_Manu, PT:= T#2S);
Enregistrement_Manu := (SEL(Enregistrement_Manu, Enregistrement_Manu, FALSE) OR TP_RAZ_Enr_Manu.Q);

(******************Gestion enregistrement des varaibles perssitantes********************************)
WritePersistentData_1(
	NETID:= '',
	PORT:= 851,
	START:= Enregistrement_Manu OR bStart,
	TMOUT:= T#1s,
	BUSY=> bBusy,
	ERR=> bError,
	ERRID=>nErrorId);
bStart := FALSE;

END_PROGRAM

// ---- POUs/Visualisation/Visu.TcPOU
PROGRAM Visu
VAR
	Info_PLC: FB_GetLocalAmsNetId;
	Start: BOOL;
	//Clignotement pour gérer des animations :
	Tmr         	: TON;   	// temporisateur On-Delay standard
    RTrig       	: R_TRIG;	// détecteur de front montant
	Tmr1         	: TON;   	// temporisateur On-Delay standard
    RTrig1       	: R_TRIG;	// détecteur de front montant
	Tmr2         	: TON;   	// temporisateur On-Delay standard
    RTrig2       	: R_TRIG;	// détecteur de front montant
	Var_Test1		: WSTRING(511);
	Var_Test2		: WSTRING;
	Var_test3		: TIME;
	Var_test4		: BOOL;
	// Gestion de l'affichage de la couleur de la cabine :	
    Opacite 		: BYTE := 66; // Opacité (0 = transparent, 255 = opaque)
	Opacite1 		: BYTE := 150; // Opacité (0 = transparent, 255 = opaque)
	//Gestion du pop-up actionneurs
	On_Off_Ventilation	:BOOL;
	//Gestion de la page Nettoyage
	Cpt_Clean		:INT;
	R_TRIG_Inc: R_TRIG;
	//Gestion de la page Recet_EnCours	
	R_TRIG_RecetEnCours: R_TRIG;
	RS_VolEau_Douche: RS;
	RS_VolEau_Lavabo: RS;
	//Gestion de la page Mode_Manu	
	R_TRIG_RecetEnCours_Manu: R_TRIG;
	RS_VolEau_Douche_Manu: RS;
	RS_VolEau_Lavabo_Manu: RS;
	Manu_Tot_Second:DINT;
	Heure_Limite_Douche:REAL;
	Minute_Limite_Douche:REAL;
	Seconde_Limite_Douche:REAL;
	Heure_Limite_Lavabo:REAL;
	Minute_Limite_Lavabo:REAL;
	Seconde_Limite_Lavabo:REAL;
	Heure_Limite_WC:REAL;
	Minute_Limite_WC:REAL;
	Seconde_Limite_WC:REAL;
	//Gestion de la page menu
	R_Trig_Init: R_TRIG;
	TON_Menu: TON;
	R_TRIG_Menu: R_TRIG;
	//Gestion des pages de pop up des alarmes avec réarmement
	NivHaut :BOOL;
	Alarms	:BOOL;
	F_TRIG_Deco: F_TRIG;
	IHM_Mesure_Debit_Deconta: REAL;
END_VAR

GVL_Visu.Page_En_Cours 	:= VisuElems.CURRENTVISU; 			// Récupération du nom de la page en cours
Var_Test1 				:= VisuElems.CurrentFullUserName;
GVL_Visu.Language 		:= VisuElems.CURRENTLANGUAGE;		// récupération du language en cours
GVL_Visu.Connexion 		:= VisuElems.CurrentUserGroupName;	// Récupération du nom de l'utilisateur en cours (Peu poser problème si plusieurs connexion en même temps)
Var_Test2 				:= VisuElems.CurrentUserName;
Var_test3 				:= VisuElems.CurrentRemainingAutoLogoutTime;
Var_test4 				:= VisuElems.CurrentUseAutoLogoutTime;
Info_PLC(bExecute:= Start, tTimeOut:= DEFAULT_ADS_TIMEOUT);

//////////////////////////////////////////////////////////////
//Gestion de la page dépollution							//
//////////////////////////////////////////////////////////////
// Mouvement de la flèche vers le haut :
IF (Mode_Cabine_Depollution)
	THEN
		GVL_Visu.Arrow_Up := GVL_Visu.Arrow_Up - 1;
		IF (GVL_Visu.Arrow_Up = 0)
			THEN
			GVL_Visu.Arrow_Up := 150;
		END_IF;
	ELSE
		GVL_Visu.Arrow_Up := 150;
END_IF
// Mouvement de la flèche vers le bas :
IF (Mode_Cabine_Depollution)
	THEN
		GVL_Visu.Arrow_Down := LIMIT(0, GVL_Visu.Arrow_Down + 1, 150);
		IF (GVL_Visu.Arrow_Down = 150)
			THEN
			GVL_Visu.Arrow_Down := 0;
		END_IF;
	ELSE
		GVL_Visu.Arrow_Down := 0;
END_IF

// Retour à la page Menu à la fin du mode Depollution
IF ((GVL_Visu.Page_En_Cours = 'Depollution') AND R_TRIG_RecetEnCours_Manu.Q)
	THEN
	VisuElems.CURRENTVISU := 'menu';
END_IF

//Affichage de la valeur de mesure
IHM_Mesure_Debit_Deconta := GVL_RegTROX.MES_RegSouf_GD_FCVT01.Mesure_EAN / LIMIT(1.0, Volume_Cabine, 1000);

//////////////////////////////////////////////////////////////
//Gestion du pop-up actionneurs								//
//////////////////////////////////////////////////////////////
IF (MES_Debit_Volh_Soufflage > 1.0)
	THEN
		On_Off_Ventilation := TRUE;
	ELSE
		On_Off_Ventilation := FALSE;
END_IF

//////////////////////////////////////////////////////////////
//Gestion de la page Nettoyage								//
//////////////////////////////////////////////////////////////
R_TRIG_Inc(CLK:= GVL_Visu.On_Off_Anim_Rap);
IF (R_TRIG_Inc.Q AND Mode_Cabine_Nettoyage)
	THEN
		Cpt_Clean := Cpt_Clean + 1;
		IF (Cpt_Clean > 7)
			THEN
				Cpt_Clean := 0;
		END_IF
END_IF
IF (NOT Mode_Cabine_Nettoyage)
	THEN
		Cpt_Clean := 0;
END_IF
CASE Cpt_Clean OF
	0:	// Etape 0 initialisation des valeurs
	GVL_Visu.Cmd_Img_Clean1 := FALSE;
	GVL_Visu.Cmd_Img_Clean2 := FALSE;
	GVL_Visu.Cmd_Img_Clean3 := FALSE;
	GVL_Visu.Cmd_Img_Clean4 := FALSE;
	GVL_Visu.Cmd_Img_Clean5 := FALSE;
	GVL_Visu.Cmd_Img_Clean6 := FALSE;
	GVL_Visu.Cmd_Img_Clean7 := FALSE;
	
	1: // Etape affichage de l'image 1
	GVL_Visu.Cmd_Img_Clean1 := TRUE;
	GVL_Visu.Cmd_Img_Clean2 := FALSE;
	GVL_Visu.Cmd_Img_Clean3 := FALSE;
	GVL_Visu.Cmd_Img_Clean4 := FALSE;
	GVL_Visu.Cmd_Img_Clean5 := FALSE;
	GVL_Visu.Cmd_Img_Clean6 := FALSE;
	GVL_Visu.Cmd_Img_Clean7 := FALSE;
	
	2: // Etape affichage de l'image 1,2
	GVL_Visu.Cmd_Img_Clean1 := TRUE;
	GVL_Visu.Cmd_Img_Clean2 := TRUE;
	GVL_Visu.Cmd_Img_Clean3 := FALSE;
	GVL_Visu.Cmd_Img_Clean4 := FALSE;
	GVL_Visu.Cmd_Img_Clean5 := FALSE;
	GVL_Visu.Cmd_Img_Clean6 := FALSE;
	GVL_Visu.Cmd_Img_Clean7 := FALSE;
	
	3: // Etape affichage de l'image 1,2,3
	GVL_Visu.Cmd_Img_Clean1 := TRUE;
	GVL_Visu.Cmd_Img_Clean2 := TRUE;
	GVL_Visu.Cmd_Img_Clean3 := TRUE;
	GVL_Visu.Cmd_Img_Clean4 := FALSE;
	GVL_Visu.Cmd_Img_Clean5 := FALSE;
	GVL_Visu.Cmd_Img_Clean6 := FALSE;
	GVL_Visu.Cmd_Img_Clean7 := FALSE;
	
	4: // Etape affichage de l'image 1,2,3,4
	GVL_Visu.Cmd_Img_Clean1 := TRUE;
	GVL_Visu.Cmd_Img_Clean2 := TRUE;
	GVL_Visu.Cmd_Img_Clean3 := TRUE;
	GVL_Visu.Cmd_Img_Clean4 := TRUE;
	GVL_Visu.Cmd_Img_Clean5 := FALSE;
	GVL_Visu.Cmd_Img_Clean6 := FALSE;
	GVL_Visu.Cmd_Img_Clean7 := FALSE;
	
	5: // Etape affichage de l'image 1,2,3,4,5
	GVL_Visu.Cmd_Img_Clean1 := TRUE;
	GVL_Visu.Cmd_Img_Clean2 := TRUE;
	GVL_Visu.Cmd_Img_Clean3 := TRUE;
	GVL_Visu.Cmd_Img_Clean4 := TRUE;
	GVL_Visu.Cmd_Img_Clean5 := TRUE;
	GVL_Visu.Cmd_Img_Clean6 := FALSE;
	GVL_Visu.Cmd_Img_Clean7 := FALSE;
	
	6: // Etape affichage de l'image 1,2,3,4,5,6
	GVL_Visu.Cmd_Img_Clean1 := TRUE;
	GVL_Visu.Cmd_Img_Clean2 := TRUE;
	GVL_Visu.Cmd_Img_Clean3 := TRUE;
	GVL_Visu.Cmd_Img_Clean4 := TRUE;
	GVL_Visu.Cmd_Img_Clean5 := TRUE;
	GVL_Visu.Cmd_Img_Clean6 := TRUE;
	GVL_Visu.Cmd_Img_Clean7 := FALSE;
	
	7: // Etape affichage de l'image 1,2,3,4,5,6,7
	GVL_Visu.Cmd_Img_Clean1 := TRUE;
	GVL_Visu.Cmd_Img_Clean2 := TRUE;
	GVL_Visu.Cmd_Img_Clean3 := TRUE;
	GVL_Visu.Cmd_Img_Clean4 := TRUE;
	GVL_Visu.Cmd_Img_Clean5 := TRUE;
	GVL_Visu.Cmd_Img_Clean6 := TRUE;
	GVL_Visu.Cmd_Img_Clean7 := TRUE;
END_CASE

// Retour à la page Menu à la fin du mode Nettoyage
IF ((GVL_Visu.Page_En_Cours = 'Nettoyage') AND R_TRIG_RecetEnCours_Manu.Q)
	THEN
	VisuElems.CURRENTVISU := 'menu';
END_IF

//////////////////////////////////////////////////////////////
//Gestion de la page Sel_Recettes							//
//////////////////////////////////////////////////////////////
IF (Nbre_Etape_Totale <> 0)
	THEN
	GVL_Visu.Visu_Btn_Start := FALSE;
	ELSE
	GVL_Visu.Visu_Btn_Start := TRUE;
END_IF

//////////////////////////////////////////////////////////////
//Gestion de la page Recet_EnCours							//
//////////////////////////////////////////////////////////////
//Affichage de la valeur du volume d'eau restant pour la douche - reset de l'affichage quand la vidange est ouverte
RS_VolEau_Douche (SET:= Mode_Auto.Mode_12 OR Mode_Auto.Mode_13, RESET1:= E_Vanne_Vidange_Douche_Ouv OR Mode_Cabine_Libre);
GVL_Visu.Visu_VolEau_Douche := Mode_Auto.Mode_12 OR Mode_Auto.Mode_13;

//Affichage de la valeur du volume d'eau restant pour le lavabo - reset de l'affichage quand la vidange est ouverte
RS_VolEau_Lavabo (SET:= Mode_Auto.Mode_14 OR Mode_Auto.Mode_15, RESET1:= E_Vanne_Vidange_Lavabo_Ouv OR Mode_Cabine_Libre);
GVL_Visu.Visu_VolEau_Lavabo := Mode_Auto.Mode_14 OR Mode_Auto.Mode_15;

//Affichage du décomptes en secondes
GVL_Visu.Visu_Tempo := Mode_Auto.Mode_1 OR Mode_Auto.Mode_2 OR Mode_Auto.Mode_4 OR Mode_Auto.Mode_5 OR Mode_Auto.Mode_6
						OR Mode_Auto.Mode_7 OR Mode_Auto.Mode_8 OR Mode_Auto.Mode_10 OR Mode_Auto.Mode_11
						OR Mode_Auto.Mode_18 OR Mode_Auto.Mode_19 OR Mode_Auto.Mode_27;

//Affichage du nombre de cycle restant de chasse d'eau
GVL_Visu.Visu_ChasseEau := Mode_Auto.Mode_9 OR Mode_Auto.Mode_26;

//Affichage du débit d'eau, peu importe si c'est la douche ou le lavabo
GVL_Visu.Visu_Debit_Eau := Mode_Auto.Mode_14 OR Mode_Auto.Mode_15 OR Mode_Auto.Mode_12 OR Mode_Auto.Mode_13;
GVL_Visu.Visu_Mes_Debit_Eau := MAX(Tab_MES_Sonde_Debit_Alim_Douche.R_MesCor,Tab_MES_Sonde_Debit_Alim_Lavabo.R_MesCor);

// Retour à la page Menu à la fin de la recette
R_TRIG_RecetEnCours(CLK:= Mode_Cabine_Libre);
IF ((GVL_Visu.Page_En_Cours = 'Recet_EnCours') AND R_TRIG_RecetEnCours.Q)
	THEN
	VisuElems.CURRENTVISU := 'menu';
END_IF

//////////////////////////////////////////////////////////////
//Gestion de la page Mode_Manu								//
//////////////////////////////////////////////////////////////
//Affichage de la valeur du volume d'eau restant pour la douche - reset de l'affichage quand la vidange est ouverte
RS_VolEau_Douche_Manu (SET:= Mode_Manu.Mode_12 OR Mode_Manu.Mode_13, RESET1:= Mode_Cabine_Libre);
GVL_Visu.Visu_VolEau_Douche_Manu := RS_VolEau_Douche_Manu.Q1;

//Affichage de la valeur du volume d'eau restant pour le lavabo - reset de l'affichage quand la vidange est ouverte
RS_VolEau_Lavabo_Manu (SET:= Mode_Manu.Mode_14 OR Mode_Manu.Mode_15, RESET1:= Mode_Cabine_Libre);
GVL_Visu.Visu_VolEau_Lavabo_Manu := RS_VolEau_Lavabo_Manu.Q1;

//Affichage du nombre de cycle restant de chasse d'eau
GVL_Visu.Visu_ChasseEau_Manu := Mode_Manu.Mode_9 OR Mode_Manu.Mode_26;

//Affichage du débit d'eau, peu importe si c'est la douche ou le lavabo
GVL_Visu.Visu_Debit_Eau_Manu := Mode_Manu.Mode_14 OR Mode_Manu.Mode_15 OR Mode_Manu.Mode_12 OR Mode_Manu.Mode_13;
GVL_Visu.Visu_Mes_Debit_Eau_Manu := MAX(Tab_MES_Sonde_Debit_Alim_Douche.R_MesCor,Tab_MES_Sonde_Debit_Alim_Lavabo.R_MesCor);

// Retour à la page Menu à la fin du mode manu
R_TRIG_RecetEnCours_Manu(CLK:= Mode_Cabine_Libre);
IF ((GVL_Visu.Page_En_Cours = 'ModeManuel') AND R_TRIG_RecetEnCours_Manu.Q)
	THEN
	VisuElems.CURRENTVISU := 'menu';
END_IF

// Conversion en integer de la variable de sélection du mode
GVL_Visu.Manu_Choix_Numero_Mode_INT := REAL_TO_INT(Manu_Choix_Numero_Mode);

// Gestion de la sélection des modes manuel présent dans le projet :
GVL_Visu.Tab_Choix_Modes[1] := FALSE;		// Mode 1 douche avec vidange avec tempo
GVL_Visu.Tab_Choix_Modes[2] := FALSE;		// Mode 2 douche sans vidange  avec tempo
GVL_Visu.Tab_Choix_Modes[3] := FALSE;		// Mode 3 douchette avec vidange
GVL_Visu.Tab_Choix_Modes[4] := TRUE;		// Mode 4 lavabo avec vidange avec tempo
GVL_Visu.Tab_Choix_Modes[5] := TRUE;		// Mode 5 lavabo sans vidange avec tempo
GVL_Visu.Tab_Choix_Modes[6] := FALSE;		// Mode 6 activation prise
GVL_Visu.Tab_Choix_Modes[7] := TRUE;		// Mode 7 vidange(s)
GVL_Visu.Tab_Choix_Modes[8] := TRUE;		// Mode 8 neutre
GVL_Visu.Tab_Choix_Modes[9] := FALSE;		// Mode 9 CHASSE D EAU GRAND VOLUME
GVL_Visu.Tab_Choix_Modes[10] := FALSE;		// Mode 10 Dépollution
GVL_Visu.Tab_Choix_Modes[11] := FALSE;		// Mode 11 bas débit
GVL_Visu.Tab_Choix_Modes[12] := FALSE;		// Mode 12 douche avec vidange transition volume d'eau
GVL_Visu.Tab_Choix_Modes[13] := FALSE;		// Mode 13 douche sans vidange transition volume d'eau
GVL_Visu.Tab_Choix_Modes[14] := TRUE;		// Mode 14 lavabo avec vidange transition volume d'eau
GVL_Visu.Tab_Choix_Modes[15] := TRUE;		// Mode 15 lavabo sans vidange transition volume d'eau
GVL_Visu.Tab_Choix_Modes[16] := FALSE;		// Mode 16 douche avec vidange avec BP
GVL_Visu.Tab_Choix_Modes[17] := FALSE;		// Mode 17 lavabo avec vidange avec BP
GVL_Visu.Tab_Choix_Modes[18] := FALSE;		// Mode 18 lavage NEP eau chaude
GVL_Visu.Tab_Choix_Modes[19] := FALSE;		// Mode 19 lavage NEP eau froide
GVL_Visu.Tab_Choix_Modes[20] := FALSE;		// Mode 20 Paramétrable (non utilisé)
GVL_Visu.Tab_Choix_Modes[21] := FALSE;		// Mode 21 alerte préparateur
GVL_Visu.Tab_Choix_Modes[22] := FALSE;		// Mode 22 alerte évaluateur
GVL_Visu.Tab_Choix_Modes[23] := FALSE;		// Mode 23 évaluation (sans moteur bypass)
GVL_Visu.Tab_Choix_Modes[24] := FALSE;		// Mode 24 évaluation (avec moteur bypass)
GVL_Visu.Tab_Choix_Modes[25] := FALSE;		// Mode 25 MISE EN CONDITION
GVL_Visu.Tab_Choix_Modes[26] := FALSE;		// Mode 26 CHASSE D EAU PETIT VOLUME
GVL_Visu.Tab_Choix_Modes[27] := FALSE;		// Mode nettoyage (version NEP)
GVL_Visu.Tab_Choix_Modes[28] := FALSE;		// Mode cabine en condition
GVL_Visu.Tab_Choix_Modes[29] := FALSE;		// Libre
GVL_Visu.Tab_Choix_Modes[30] := FALSE;		// Mode 30 à 59 texte éditable
//premier mode
GVL_Visu.Min_Mode_Manu := 4;
//dernier mode
GVL_Visu.Max_Mode_Manu := 15;

//Affichage du paramétrage du débit d'eau Lavabo
GVL_Visu.Affich_Debit_Eau_Manu := (Manu_Choix_Numero_Mode = 14) OR (Manu_Choix_Numero_Mode = 15)
											OR (Manu_Choix_Numero_Mode = 12) OR (Manu_Choix_Numero_Mode = 13);
//Affichage du paramétrage du débit d'eau douche
GVL_Visu.Affich_Debit_Eau_Manu_Douche := (Manu_Choix_Numero_Mode = 12) OR (Manu_Choix_Numero_Mode = 13);
//Affichage du paramétrage du débit d'eau Lavabo
GVL_Visu.Affich_Debit_Eau_Manu_Lavabo := (Manu_Choix_Numero_Mode = 14) OR (Manu_Choix_Numero_Mode = 15);

//Affichage de la consigne de température
GVL_Visu.Visu_Temp_Manu := 	Option_Regul_Temp_Eau AND
							((Manu_Choix_Numero_Mode = 1) OR (Manu_Choix_Numero_Mode = 2)
							OR (Manu_Choix_Numero_Mode = 4) OR (Manu_Choix_Numero_Mode = 5)
							OR (Manu_Choix_Numero_Mode = 12) OR (Manu_Choix_Numero_Mode = 13)
							OR (Manu_Choix_Numero_Mode = 14) OR (Manu_Choix_Numero_Mode = 15));								
									
//Affichage du paramétrage de la chasse d'eau
GVL_Visu.Affich_ChasseEau_Manu := (Manu_Choix_Numero_Mode = 9) OR (Manu_Choix_Numero_Mode = 26);

//Gestion des limites minimum et maximum du volume d'eau lors d'une vidange fermée
IF (Manu_Choix_Numero_Mode = 13)		//Douche
	THEN
	Manu_Lct_Cons_Vol_Douche := LIMIT(0, Manu_Lct_Cons_Vol_Douche, Volume_Secu_Debord_Douche);
	ELSE
	Manu_Lct_Cons_Vol_Douche := LIMIT(0, Manu_Lct_Cons_Vol_Douche, 999);
END_IF
IF (Manu_Choix_Numero_Mode = 15)		//Lavabo
	THEN
	Manu_Lct_Cons_Vol_Lavabo := LIMIT(0, Manu_Lct_Cons_Vol_Lavabo, Volume_Secu_Debord_Lavabo);
	ELSE
	Manu_Lct_Cons_Vol_Lavabo := LIMIT(0, Manu_Lct_Cons_Vol_Lavabo, 999);
END_IF

//Gestion des limites de temporisation lors d'une vidange fermée et du temps de remplissage du WC
Manu_Tot_Second := (TO_DINT(Manu_Tempo_Transition_Heure) * 3600)
					+ (TO_DINT(Manu_Tempo_Transition_Minute) * 60)
					+ (TO_DINT(Manu_Tempo_Transition_Seconde));
//Limite de la sécurité haute de la douche
Seconde_Limite_Douche 	:= TO_REAL((Temp_Secu_Debord_Douche) MOD 60);
Minute_Limite_Douche 	:= TO_REAL((Temp_Secu_Debord_Douche / 60) MOD 60);
Heure_Limite_Douche 	:= TO_REAL((Temp_Secu_Debord_Douche / 3600) MOD 24);
//Limite de la sécurité haute du lavabo
Seconde_Limite_Lavabo	:= TO_REAL((Temp_Secu_Debord_Lavabo) MOD 60);
Minute_Limite_Lavabo 	:= TO_REAL((Temp_Secu_Debord_Lavabo / 60) MOD 60);
Heure_Limite_Lavabo 	:= TO_REAL((Temp_Secu_Debord_Lavabo / 3600) MOD 24);
//Limite de la sécurité haute du cycle de chasse d'eau
Seconde_Limite_WC		:= TO_REAL((Temps_Remplissage_WC) MOD 60);
Minute_Limite_WC 		:= TO_REAL((Temps_Remplissage_WC / 60) MOD 60);
Heure_Limite_WC 		:= TO_REAL((Temps_Remplissage_WC / 3600) MOD 24);
IF (Manu_Choix_Numero_Mode = 2 AND Option_Douche)
	THEN	//Douche
	IF (Manu_Tot_Second > TO_DINT(Temp_Secu_Debord_Douche))
		THEN
		Manu_Tempo_Transition_Seconde := Seconde_Limite_Douche;
		Manu_Tempo_Transition_Minute := Minute_Limite_Douche;
		Manu_Tempo_Transition_Heure := Heure_Limite_Douche;
	END_IF
	ELSIF (Manu_Choix_Numero_Mode = 5 AND Option_Lavabo)
	THEN	//Lavabo
	IF (Manu_Tot_Second > TO_DINT(Temp_Secu_Debord_Lavabo))
		THEN
		Manu_Tempo_Transition_Seconde := Seconde_Limite_Lavabo;
		Manu_Tempo_Transition_Minute := Minute_Limite_Lavabo;
		Manu_Tempo_Transition_Heure := Heure_Limite_Lavabo;
	END_IF
	ELSIF (Manu_Choix_Numero_Mode = 9 OR Manu_Choix_Numero_Mode = 26 AND (Option_WC_GV OR Option_WC_PV))
	THEN	//WC
	IF (Manu_Tot_Second > TO_DINT(Temps_Remplissage_WC))
		THEN
		Manu_Tempo_Transition_Seconde := Seconde_Limite_WC;
		Manu_Tempo_Transition_Minute := Minute_Limite_WC;
		Manu_Tempo_Transition_Heure := Heure_Limite_WC;
	END_IF
	ELSE
	Manu_Tempo_Transition_Seconde := Manu_Tempo_Transition_Seconde;
	Manu_Tempo_Transition_Minute := Manu_Tempo_Transition_Minute;
	Manu_Tempo_Transition_Heure := Manu_Tempo_Transition_Heure;
END_IF

//////////////////////////////////////////////////////////////
//gestion de la page menu									//
//////////////////////////////////////////////////////////////
//Initialisation des Enbale forçage lors du retour sur la page menu
R_Trig_Init(CLK:= (GVL_Visu.Page_En_Cours = 'menu'));
IF(R_Trig_Init.Q)
	THEN
	EF_Cmd_PC_Cab  							:= FALSE;
	EF_Cmd_Vanne_Alim_Douche  				:= FALSE;
	EF_Cmd_Vanne_Alim_Douchette  			:= FALSE;
	EF_Cmd_Vanne_Alim_Lavabo  				:= FALSE;
	EF_Cmd_Vanne_Vid_Douche  				:= FALSE;
	EF_Cmd_Vanne_Vid_Lavabo 				:= FALSE;
	EF_Cmd_ElectroValve_Alim_Douche  		:= FALSE;
	EF_Cmd_ElectroValve_Alim_Lavabo 		:= FALSE;
	EF_Cons_Registre_Extraction 			:= FALSE;
	EF_Cons_Registre_Soufflage 				:= FALSE;
	EF_Vanne_Souf_Bas_Deb 					:= FALSE;
	EF_Vanne_Ext_Bas_Deb 					:= FALSE;
	EF_Cons_Reg_Etanche_Ext 				:= FALSE;
	EF_Cmd_Reg_Etanche_Souf 				:= FALSE;
	EF_Cons_V3V_Eau_Mitig 					:= FALSE;
	EF_Vanne_Alim_NEP 						:= FALSE;
	EF_Cons_V3V_Bat_Froid_CTA  				:= FALSE;
	EF_Cmd_Verin_WC_GV  					:= FALSE;
	EF_Cmd_Verin_WC_PV  					:= FALSE;
	Tab_MotRep_CTA.Mot_Ecriture.0			:= FALSE;
	Tab_MotSouf_CTA.Mot_Ecriture.0			:= FALSE;
	Tab_Mot_Aerobox_Bas_Deb.Mot_Ecriture.0	:= FALSE;
	Tab_Mot_ByPass.Mot_Ecriture.0			:= FALSE;
END_IF

(*//Gestion du retour sur la page 'Accueil' après un certain délais sur la page Menu
TON_Menu(IN:= (GVL_Visu.Page_En_Cours = 'menu'), PT:= T#10M);
R_TRIG_Menu(CLK:= TON_Menu.Q);
IF (R_TRIG_Menu.Q)
	THEN
	VisuElems.CURRENTVISU := 'Accueil';
END_IF*)

//////////////////////////////////////////////////////////////
//Gestion des pages de pop up des alarmes avec réarmement	//
//////////////////////////////////////////////////////////////
NivHaut := 	Defaut_Debordement_Douche OR Defaut_Debordement_Lavabo;
Alarms	:= 	NOT NivHaut AND Condi_Affich_Rearm;
GVL_Visu.Affichage_PopUp_HightLevel	:= NivHaut;
GVL_Visu.Affichage_PopUp_Alarm := Alarms;

//////////////////////////////////////////////////////////////
//Autres													//
//////////////////////////////////////////////////////////////	
//Clignotement lent pour gérer des animations :
Tmr(IN := TRUE, PT := T#500MS);
RTrig(CLK := Tmr.Q);
IF RTrig.Q THEN
    GVL_Visu.On_Off_Anim := NOT GVL_Visu.On_Off_Anim;  	// bascule ON↔OFF
    Tmr(IN := FALSE);                					// arrêt court du timer pour le remettre à zéro
END_IF
IF NOT Tmr.Q THEN
    Tmr(IN := TRUE);
END_IF
//Clignotement rapide pour gérer des animations :
Tmr1(IN := TRUE, PT := T#200MS);
RTrig1(CLK := Tmr1.Q);
IF RTrig1.Q THEN
    GVL_Visu.On_Off_Anim_Rap := NOT GVL_Visu.On_Off_Anim_Rap;  	// bascule ON↔OFF
    Tmr1(IN := FALSE);                					// arrêt court du timer pour le remettre à zéro
END_IF
IF NOT Tmr1.Q THEN
    Tmr1(IN := TRUE);
END_IF
//Clignotement rapide pour gérer des animations :
Tmr2(IN := TRUE, PT := T#1S);
RTrig2(CLK := Tmr2.Q);
IF RTrig2.Q THEN
    GVL_Visu.On_Off_Anim_Lent := NOT GVL_Visu.On_Off_Anim_Lent;  	// bascule ON↔OFF
    Tmr2(IN := FALSE);                					// arrêt court du timer pour le remettre à zéro
END_IF
IF NOT Tmr2.Q THEN
    Tmr2(IN := TRUE);
END_IF

// Sélection de l'affichage du numéro de la cabine sur les visuels :
CASE GVL_Visu.Numero_Cabine OF
	0: GVL_Visu.Nom_Cabine_FR := 'PAS DE NOM'; GVL_Visu.Nom_Cabine_EN := 'NO NAME';
	1: GVL_Visu.Nom_Cabine_FR := 'CABINE 1'; GVL_Visu.Nom_Cabine_EN := 'BOOTH 1';
	2: GVL_Visu.Nom_Cabine_FR := 'CABINE 2'; GVL_Visu.Nom_Cabine_EN := 'BOOTH 2';
	3: GVL_Visu.Nom_Cabine_FR := 'CABINE 3'; GVL_Visu.Nom_Cabine_EN := 'BOOTH 3';
	4: GVL_Visu.Nom_Cabine_FR := 'CABINE 4'; GVL_Visu.Nom_Cabine_EN := 'BOOTH 4';
	5: GVL_Visu.Nom_Cabine_FR := 'CABINE 5'; GVL_Visu.Nom_Cabine_EN := 'BOOTH 5';
	6: GVL_Visu.Nom_Cabine_FR := 'CABINE 6'; GVL_Visu.Nom_Cabine_EN := 'BOOTH 6';
	7: GVL_Visu.Nom_Cabine_FR := 'CABINE 7'; GVL_Visu.Nom_Cabine_EN := 'BOOTH 7';
	8: GVL_Visu.Nom_Cabine_FR := 'CABINE 8'; GVL_Visu.Nom_Cabine_EN := 'BOOTH 8';
	9: GVL_Visu.Nom_Cabine_FR := 'CABINE 9'; GVL_Visu.Nom_Cabine_EN := 'BOOTH 9';
	10: GVL_Visu.Nom_Cabine_FR := 'CABINE 10'; GVL_Visu.Nom_Cabine_EN := 'BOOTH 10';
	11: GVL_Visu.Nom_Cabine_FR := 'CABINE 11'; GVL_Visu.Nom_Cabine_EN := 'BOOTH 11';
	12: GVL_Visu.Nom_Cabine_FR := 'CABINE 12'; GVL_Visu.Nom_Cabine_EN := 'BOOTH 12';
	13: GVL_Visu.Nom_Cabine_FR := 'CABINE 13'; GVL_Visu.Nom_Cabine_EN := 'BOOTH 13';
	14: GVL_Visu.Nom_Cabine_FR := 'CABINE 14'; GVL_Visu.Nom_Cabine_EN := 'BOOTH 14';
	15: GVL_Visu.Nom_Cabine_FR := 'CABINE 15'; GVL_Visu.Nom_Cabine_EN := 'BOOTH 15';
	16: GVL_Visu.Nom_Cabine_FR := 'CABINE 16'; GVL_Visu.Nom_Cabine_EN := 'BOOTH 16';
	17: GVL_Visu.Nom_Cabine_FR := 'CABINE 17'; GVL_Visu.Nom_Cabine_EN := 'BOOTH 17';
	18: GVL_Visu.Nom_Cabine_FR := 'CABINE 18'; GVL_Visu.Nom_Cabine_EN := 'BOOTH 18';
	19: GVL_Visu.Nom_Cabine_FR := 'CABINE 19'; GVL_Visu.Nom_Cabine_EN := 'BOOTH 19';
	20: GVL_Visu.Nom_Cabine_FR := 'CABINE 20'; GVL_Visu.Nom_Cabine_EN := 'BOOTH 20';
END_CASE

// Gestion de la connexion de l'utilisateur Admin :
IF (GVL_Visu.Connexion = "Admin") THEN GVL_Visu.Etat_Connexion := TRUE; ELSE GVL_Visu.Etat_Connexion := FALSE; END_IF;

//Gestion du retour à la pague menu si déconnexion
F_TRIG_Deco(CLK:= GVL_Visu.Etat_Connexion);
IF(F_TRIG_Deco.Q) THEN
	VisuElems.CURRENTVISU := 'menu';
END_IF

// Gestion de l'affichage de la couleur de la cabine :
GVL_Visu.Couleur_Cabine := SHL(TO_DWORD(Opacite), 24) OR SHL(TO_DWORD(Cde_Rouge_Cabine), 16) OR SHL(TO_DWORD(Cde_Vert_Cabine), 8) OR TO_DWORD(Cde_Bleu_Cabine);
GVL_Visu.Couleur_Cabine2 := SHL(TO_DWORD(Opacite1), 24) OR SHL(TO_DWORD(Cde_Rouge_Cabine), 16) OR SHL(TO_DWORD(Cde_Vert_Cabine), 8) OR TO_DWORD(Cde_Bleu_Cabine);

// Gestion du changement de page automatique si on es sur la page menu et qu'il y'a un mode en cours (depo, auto, manu, net)
IF(Mode_Cabine_Automatique)
	THEN
	VisuElems.CURRENTVISU := 'Recet_EnCours';
END_IF
IF(NOT Mode_Cabine_Automatique AND Mode_Cabine_Manuel)
	THEN
	VisuElems.CURRENTVISU := 'ModeManuel';
END_IF
IF(NOT Mode_Cabine_Automatique AND Mode_Cabine_Nettoyage)
	THEN
	VisuElems.CURRENTVISU := 'Nettoyage';
END_IF
IF(NOT Mode_Cabine_Automatique AND Mode_Cabine_Depollution)
	THEN
	VisuElems.CURRENTVISU := 'Depollution';
END_IF

END_PROGRAM

// ---- POUs/Visualisation/Alarmes.TcPOU
PROGRAM Alarmes
VAR
	NB_ALARMES_MAX      : UINT := 100;
    GA_Alarmes        	: ARRAY[1..2, 1..100] OF ST_Alarmes;
    GA_AlarmesActives 	: ARRAY[1..2, 1..100] OF ST_Alarmes;
	Tab_Alarme_FREN		: ARRAY[1..2, 1..100] OF STRING(80);
    G_NbAlarmesActives  : UINT := 0;
	
	i         : UINT;
    idx       : UINT 	:= 0;
END_VAR

//////////////////////////////////////////////////////////////
// gestion des alarmes (bilingue FR/EN)                     //
//////////////////////////////////////////////////////////////
//Déclaration des alarmes
//Alarme 1
GA_Alarmes[1, 1].Id := 1;
GA_Alarmes[1, 1].Libelle := 'Défaut débordement de la douche / à réarmer';
GA_Alarmes[2, 1].Libelle := 'High water level in shower tray detected / must be acquit !';
GA_Alarmes[1, 1].Active := Defaut_Debordement_Douche;

//Alarme 2
GA_Alarmes[1, 2].Id := 2;
GA_Alarmes[1, 2].Libelle := 'Défaut débordement du lavabo / à réarmer';
GA_Alarmes[2, 2].Libelle := 'High water level in sink tray detected / must be acquit !';
GA_Alarmes[1, 2].Active := Defaut_Debordement_Lavabo;

//Alarme 3
GA_Alarmes[1, 3].Id := 3;
GA_Alarmes[1, 3].Libelle := 'Défaut discordance débit d’eau de la douche / à réarmer';
GA_Alarmes[2, 3].Libelle := 'Mismatch in shower water flow rate / must be acquit !';
GA_Alarmes[1, 3].Active := Defaut_Discord_Deb_Eau_Douche;

//Alarme 4
GA_Alarmes[1, 4].Id := 4;
GA_Alarmes[1, 4].Libelle := 'Défaut discordance débit d’eau du lavabo / à réarmer';
GA_Alarmes[2, 4].Libelle := 'Mismatch in sink water flow rate / must be acquit !';
GA_Alarmes[1, 4].Active := Defaut_Discord_Deb_Eau_Lavabo;

//Alarme 5
GA_Alarmes[1, 5].Id := 5;
GA_Alarmes[1, 5].Libelle := 'Défaut discordance prise de courant / à réarmer';
GA_Alarmes[2, 5].Libelle := 'Power plug supply mismatch / must be acquit !';
GA_Alarmes[1, 5].Active := Defaut_Discord_PC_Cab;

//Alarme 6
GA_Alarmes[1, 6].Id := 6;
GA_Alarmes[1, 6].Libelle := 'Défaut prise forcée manuellement / à réarmer';
GA_Alarmes[2, 6].Libelle := 'Manually forced power plug / must be acquit !';
GA_Alarmes[1, 6].Active := Def_Discord_Alim_Prise;

//Alarme 7
GA_Alarmes[1, 7].Id := 7;
GA_Alarmes[1, 7].Libelle := 'Défaut prise lors de l’ouverture porte / à réarmer';
GA_Alarmes[2, 7].Libelle := 'Door open during a power plug cycle / must be acquit !';
GA_Alarmes[1, 7].Active := Def_Prise_Porte_Ouverte;

//Alarme 8
GA_Alarmes[1, 8].Id := 8;
GA_Alarmes[1, 8].Libelle := 'Défaut pompe de relevage / à réarmer';
GA_Alarmes[2, 8].Libelle := 'Error on the lifting pump / must be acquit !';
GA_Alarmes[1, 8].Active := Defaut_Pompe_Relevage;

//Alarme 9
GA_Alarmes[1, 9].Id := 9;
GA_Alarmes[1, 9].Libelle := 'Défaut porte ouverte depuis plus d une minute';
GA_Alarmes[2, 9].Libelle := 'Door open for more than one minute';
GA_Alarmes[1, 9].Active := Defaut_Porte_Ouverte;

//Alarme 10
GA_Alarmes[1, 10].Id := 10;
GA_Alarmes[1, 10].Libelle := 'Défaut de communication avec la passerelle LED';
GA_Alarmes[2, 10].Libelle := 'Light gateway communication error';
GA_Alarmes[1, 10].Active := Defaut_Com_Dalcnet;

//Alarme 11
GA_Alarmes[1, 11].Id := 11;
GA_Alarmes[1, 11].Libelle := 'Défaut de communication avec la vanne thermostatique de la cabine';
GA_Alarmes[2, 11].Libelle := 'thermostatic valve gateway communication error';
GA_Alarmes[1, 11].Active := Defaut_Com_Vanne_General;

//Alarme 12
GA_Alarmes[1, 12].Id := 12;
GA_Alarmes[1, 12].Libelle := 'Défaut de communication avec la vanne thermostatique générale';
GA_Alarmes[2, 12].Libelle := 'thermostatic valve gateway communication error';
GA_Alarmes[1, 12].Active := Defaut_Com_Vanne_General;

//Alarme 13
GA_Alarmes[1, 13].Id := 13;
GA_Alarmes[1, 13].Libelle := 'Défaut de communication avec l’automate maitre';
GA_Alarmes[2, 13].Libelle := 'Master PLC communication error';
GA_Alarmes[1, 13].Active := Defaut_Com_Client;

//Alarme 14
GA_Alarmes[1, 14].Id := 14;
GA_Alarmes[1, 14].Libelle := 'Discordance ouverture de la vanne de vidange de la douche';
GA_Alarmes[2, 14].Libelle := 'Water drain shower valve fault - not opened';
GA_Alarmes[1, 14].Active := Defaut_Discord_Vanne_Vid_Douche_Ouv;

//Alarme 15
GA_Alarmes[1, 15].Id := 15;
GA_Alarmes[1, 15].Libelle := 'Discordance fermeture de la vanne de vidange de la douche';
GA_Alarmes[2, 15].Libelle := 'Water drain shower valve fault - not closed';
GA_Alarmes[1, 15].Active := Defaut_Discord_Vanne_Vid_Douche_Ferm;

//Alarme 16
GA_Alarmes[1, 16].Id := 16;
GA_Alarmes[1, 16].Libelle := 'Discordance ouverture de la vanne de vidange du lavabo';
GA_Alarmes[2, 16].Libelle := 'Water drain sink valve fault - not opened';
GA_Alarmes[1, 16].Active := Defaut_Discord_Vanne_Vid_Lavabo_Ouv;

//Alarme 17
GA_Alarmes[1, 17].Id := 17;
GA_Alarmes[1, 17].Libelle := 'Discordance fermeture de la vanne de vidange du lavabo';
GA_Alarmes[2, 17].Libelle := 'Water drain sink valve fault - not closed';
GA_Alarmes[1, 17].Active := Defaut_Discord_Vanne_Vid_Lavabo_Ferm;

//Alarme 18
GA_Alarmes[1, 18].Id := 18;
GA_Alarmes[1, 18].Libelle := 'Discordance ouverture de la vanne d’alimentation de la douche';
GA_Alarmes[2, 18].Libelle := 'Water supply shower valve fault - not opened';
GA_Alarmes[1, 18].Active := Defaut_Discord_Vanne_Alim_Douche_Ouv;

//Alarme 19
GA_Alarmes[1, 19].Id := 19;
GA_Alarmes[1, 19].Libelle := 'Discordance fermeture de la vanne d alimentation de la douche';
GA_Alarmes[2, 19].Libelle := 'Water supply shower valve fault - not closed';
GA_Alarmes[1, 19].Active := Defaut_Discord_Vanne_Alim_Douche_Ferm;

//Alarme 20
GA_Alarmes[1, 20].Id := 20;
GA_Alarmes[1, 20].Libelle := 'Discordance ouverture de la vanne d’alimentation du lavabo';
GA_Alarmes[2, 20].Libelle := 'Water supply sink valve fault - not opened';
GA_Alarmes[1, 20].Active := Defaut_Discord_Vanne_Alim_Lavabo_Ouv;

//Alarme 21
GA_Alarmes[1, 21].Id := 21;
GA_Alarmes[1, 21].Libelle := 'Discordance fermeture de la vanne d’alimentation du lavabo';
GA_Alarmes[2, 21].Libelle := 'Water supply sink valve fault - not closed';
GA_Alarmes[1, 21].Active := Defaut_Discord_Vanne_Alim_Lavabo_Ferm;

//Alarme 22
GA_Alarmes[1, 22].Id := 22;
GA_Alarmes[1, 22].Libelle := 'Discordance ouverture de la vanne d’alimentation de la douchette';
GA_Alarmes[2, 22].Libelle := 'Water supply handspray valve fault - not opened';
GA_Alarmes[1, 22].Active := Defaut_Discord_Vanne_Alim_Douchette_Ouv;

//Alarme 23
GA_Alarmes[1, 23].Id := 23;
GA_Alarmes[1, 23].Libelle := 'Discordance fermeture de la vanne d’alimentation de la douchette';
GA_Alarmes[2, 23].Libelle := 'Water supply handspray valve fault - not closed';
GA_Alarmes[1, 23].Active := Defaut_Discord_Vanne_Alim_Douchette_Ferm;

//Alarme 24
GA_Alarmes[1, 24].Id := 24;
GA_Alarmes[1, 24].Libelle := 'Discordance ouverture vanne alimentation NEP';
GA_Alarmes[2, 24].Libelle := 'Mismatch between CIP supply valve opening';
GA_Alarmes[1, 24].Active := Defaut_Discord_Vanne_Alim_NEP_Ouv;

//Alarme 25
GA_Alarmes[1, 25].Id := 25;
GA_Alarmes[1, 25].Libelle := 'Discordance fermeture vanne alimentation NEP';
GA_Alarmes[2, 25].Libelle := 'Mismatch between CIP supply valve closure';
GA_Alarmes[1, 25].Active := Defaut_Discord_Vanne_Alim_NEP_Ferm;

//Alarme 26
GA_Alarmes[1, 26].Id := 26;
GA_Alarmes[1, 26].Libelle := 'Discordance ouverture de la vanne de soufflage bas débit';
GA_Alarmes[2, 26].Libelle := 'Air supply low flow valve fault - not opened';
GA_Alarmes[1, 26].Active := Defaut_Discord_Vanne_Souf_Bas_Deb_Ouv;

//Alarme 27
GA_Alarmes[1, 27].Id := 27;
GA_Alarmes[1, 27].Libelle := 'Discordance fermeture de la vanne de soufflage bas débit';
GA_Alarmes[2, 27].Libelle := 'Air supply low flow valve fault - not closed';
GA_Alarmes[1, 27].Active := Defaut_Discord_Vanne_Souf_Bas_Deb_Ferm;

//Alarme 28
GA_Alarmes[1, 28].Id := 28;
GA_Alarmes[1, 28].Libelle := 'Discordance ouverture de la vanne d’extraction bas débit';
GA_Alarmes[2, 28].Libelle := 'Exhaust low flow valve fault - not opened';
GA_Alarmes[1, 28].Active := Defaut_Discord_Vanne_Ext_Bas_Deb_Ouv;

//Alarme 29
GA_Alarmes[1, 29].Id := 29;
GA_Alarmes[1, 29].Libelle := 'Discordance fermeture de la vanne d’extraction bas débit';
GA_Alarmes[2, 29].Libelle := 'Exhaust low flow valve fault - not closed';
GA_Alarmes[1, 29].Active := Defaut_Discord_Vanne_Ext_Bas_Deb_Ferm;

//Alarme 30
GA_Alarmes[1, 30].Id := 30;
GA_Alarmes[1, 30].Libelle := 'Discordance de régulation du débit d’extraction';
GA_Alarmes[2, 30].Libelle := 'Exhaust flow regulation fault';
GA_Alarmes[1, 30].Active := Defaut_Discord_Deb_Ext;

//Alarme 31
GA_Alarmes[1, 31].Id := 31;
GA_Alarmes[1, 31].Libelle := 'Discordance de régulation du débit de soufflage';
GA_Alarmes[2, 31].Libelle := 'Supply flow regulation fault';
GA_Alarmes[1, 31].Active := Defaut_Discord_Deb_Souf;

//Alarme 32
GA_Alarmes[1, 32].Id := 32;
GA_Alarmes[1, 32].Libelle := 'Défaut différentiel prise électrique';
GA_Alarmes[2, 32].Libelle := 'Differential fault in electrical outlet';
GA_Alarmes[1, 32].Active := Defaut_Differentiel_Prise_Elec;

//Alarme 33
GA_Alarmes[1, 33].Id := 33;
GA_Alarmes[1, 33].Libelle := 'Registre d’extraction non fermé';
GA_Alarmes[2, 33].Libelle := 'Booth air exhaust damper no closed';
GA_Alarmes[1, 33].Active := Defaut_Discord_Reg_Ext_Ferm;

//Alarme 34
GA_Alarmes[1, 34].Id := 34;
GA_Alarmes[1, 34].Libelle := 'Registre de soufflage non fermé';
GA_Alarmes[2, 34].Libelle := 'Booth air supply damper no closed';
GA_Alarmes[1, 34].Active := Defaut_Discord_Reg_Souf_Ferm;

//Alarme 35
GA_Alarmes[1, 35].Id := 35;
GA_Alarmes[1, 35].Libelle := 'Défaut Klixon batterie électrique';
GA_Alarmes[2, 35].Libelle := 'Electric battery klixon fault';
GA_Alarmes[1, 35].Active := Defaut_Klixon_BattElec;

//Alarme 36
GA_Alarmes[1, 36].Id := 36;
GA_Alarmes[1, 36].Libelle := 'Discordance ouverture du registre d’extraction';
GA_Alarmes[2, 36].Libelle := 'Discordance opening of the exhaust damper';
GA_Alarmes[1, 36].Active := Defaut_Discord_Reg_Etanche_Ext;

//Alarme 37
GA_Alarmes[1, 37].Id := 37;
GA_Alarmes[1, 37].Libelle := 'Défaut discordance de régulation de pression';
GA_Alarmes[2, 37].Libelle := 'Pressure regulation mismatch';
GA_Alarmes[1, 37].Active := Defaut_Discord_Regul_Press_Cab;

//Alarme 38
GA_Alarmes[1, 38].Id := 38;
GA_Alarmes[1, 38].Libelle := 'Défaut de communication avec le registre de soufflage';
GA_Alarmes[2, 38].Libelle := 'Communication failure with the supply air damper';
GA_Alarmes[1, 38].Active := Defaut_Com_Reg_Souf;

//Alarme 39
GA_Alarmes[1, 39].Id := 39;
GA_Alarmes[1, 39].Libelle := 'Défaut de communication avec le registre d’extraction';
GA_Alarmes[2, 39].Libelle := 'Communication failure with the exhaust damper';
GA_Alarmes[1, 39].Active := Defaut_Com_Reg_Ext;

//Alarme 40
GA_Alarmes[1, 40].Id := 40;
GA_Alarmes[1, 40].Libelle := 'Défaut avec le module bas débit';
GA_Alarmes[2, 40].Libelle := 'Fault with the low flow module';
GA_Alarmes[1, 40].Active := Defaut_Ensemble_Bas_Debit;

//Alarme 41
GA_Alarmes[1, 41].Id := 41;
GA_Alarmes[1, 41].Libelle := 'Défaut avec le module Bypass';
GA_Alarmes[2, 41].Libelle := 'Fault with the Bypass module';
GA_Alarmes[1, 41].Active := Defaut_Ensemble_Bypass;

//Alarme 42
GA_Alarmes[1, 42].Id := 42;
GA_Alarmes[1, 42].Libelle := 'Défaut capteur de pression de la cabine';
GA_Alarmes[2, 42].Libelle := 'Booth pressure sensor fault';
GA_Alarmes[1, 42].Active := Defaut_Sonde_Press_Cabine;

//Alarme 43
GA_Alarmes[1, 43].Id := 43;
GA_Alarmes[1, 43].Libelle := 'Défaut capteur de température de la cabine';
GA_Alarmes[2, 43].Libelle := 'Booth temperature sensor fault';
GA_Alarmes[1, 43].Active := Defaut_Sonde_Temp_Cabine;

//Alarme 44
GA_Alarmes[1, 44].Id := 44;
GA_Alarmes[1, 44].Libelle := 'Défaut capteur d’hygrométrie de la cabine';
GA_Alarmes[2, 44].Libelle := 'Booth humidity sensor fault';
GA_Alarmes[1, 44].Active := Defaut_Sonde_Hygro_Cabine;

//Alarme 45
GA_Alarmes[1, 45].Id := 45;
GA_Alarmes[1, 45].Libelle := 'Défaut capteur température eau mitigée';
GA_Alarmes[2, 45].Libelle := 'Mixed water temperature sensor fault';
GA_Alarmes[1, 45].Active := Defaut_Sonde_Temp_Eau_Mitig;

//Alarme 46
GA_Alarmes[1, 46].Id := 46;
GA_Alarmes[1, 46].Libelle := 'Defaut sur le moteur de soufflage de la CTA climatique';
GA_Alarmes[2, 46].Libelle := 'Fault on air supply motor of climatic AHU';
GA_Alarmes[1, 46].Active := Defaut_MotSouf_CTA;

//Alarme 47
GA_Alarmes[1, 47].Id := 47;
GA_Alarmes[1, 47].Libelle := 'Defaut sur le moteur de reprise de la CTA climatique';
GA_Alarmes[2, 47].Libelle := 'Fault on air return motor of climatic AHU';
GA_Alarmes[1, 47].Active := Defaut_MotRep_CTA;

//Alarme 48
GA_Alarmes[1, 48].Id := 48;
GA_Alarmes[1, 48].Libelle := 'Defaut seuil haut d’hygrométrie de soufflage de la CTA climatique';
GA_Alarmes[2, 48].Libelle := 'High humidity threshold fault in the supply air of climatic AHU';
GA_Alarmes[1, 48].Active := Defaut_Hygrostat_CTA;

//Alarme 49
GA_Alarmes[1, 49].Id := 49;
GA_Alarmes[1, 49].Libelle := 'Defaut alimentation de la batterie electrique de la CTA climatique';
GA_Alarmes[2, 49].Libelle := 'Power supply failure of the electric battery of climatic AHU';
GA_Alarmes[1, 49].Active := Defaut_Alim_BatElec_CTA;
//Alarme 50
GA_Alarmes[1, 50].Id := 50;
GA_Alarmes[1, 50].Libelle := 'Defaut sur l’humidificateur de la CTA climatique';
GA_Alarmes[2, 50].Libelle := 'Fault on humidifier of climatic AHU';
GA_Alarmes[1, 50].Active := Defaut_Humi_CTA;

//Alarme 51
GA_Alarmes[1, 51].Id := 51;
GA_Alarmes[1, 51].Libelle := 'Defaut de discordance sur la régulation de la température';
GA_Alarmes[2, 51].Libelle := 'Mismatch with the temperature control of the booth';
GA_Alarmes[1, 51].Active := Defaut_Regul_Temp;

//Alarme 52
GA_Alarmes[1, 52].Id := 52;
GA_Alarmes[1, 52].Libelle := 'Défaut de discordance sur la régulation d’hygrométrie';
GA_Alarmes[2, 52].Libelle := 'Mismatch with the hygrometer control of the booth';
GA_Alarmes[1, 52].Active := Defaut_Regul_Hygro;

//Alarme 53
GA_Alarmes[1, 53].Id := 53;
GA_Alarmes[1, 53].Libelle := 'Défaut temperature de soufflage CTA climatique trop haute';
GA_Alarmes[2, 53].Libelle := 'Faulty supply air temperature AHU climatic too high';
GA_Alarmes[1, 53].Active := Defaut_Thermostat_Secu;

//Alarme 54
GA_Alarmes[1, 54].Id := 54;
GA_Alarmes[1, 54].Libelle := 'Défaut sonde de température soufflage CTA climatique';
GA_Alarmes[2, 54].Libelle := 'Faulty supply air temperature sensor in AHU Climatic';
GA_Alarmes[1, 54].Active := Defaut_Sonde_Temp_Souf;

//Alarme 55
GA_Alarmes[1, 55].Id := 55;
GA_Alarmes[1, 55].Libelle := 'Défaut discordance du soufflage de la CTA climatique';
GA_Alarmes[2, 55].Libelle := 'Mismatch in the airflow of the AHU Climatic';
GA_Alarmes[1, 55].Active := Defaut_Discord_Souf_CTA;

//Alarme 56
GA_Alarmes[1, 56].Id := 56;
GA_Alarmes[1, 56].Libelle := 'Défaut communication du Registre de soufflage gros débit';
GA_Alarmes[2, 56].Libelle := 'High-flow blow damper communication fault';
GA_Alarmes[1, 56].Active := GVL_RegTROX.RegSouf_GD_FCVT01_DefCom;

//Alarme 57
GA_Alarmes[1, 57].Id := 57;
GA_Alarmes[1, 57].Libelle := 'Défaut discordance débit du Registre de soufflage gros débit';
GA_Alarmes[2, 57].Libelle := 'Mismatch Flow Rate of High Flow Blow damper';
GA_Alarmes[1, 57].Active := GVL_RegTROX.RegSouf_GD_FCVT01_Def_DiscordDeb;

//Alarme 58
GA_Alarmes[1, 58].Id := 58;
GA_Alarmes[1, 58].Libelle := 'Défaut communication du Registre de soufflage petit débit';
GA_Alarmes[2, 58].Libelle := 'Low-flow blow damper communication fault';
GA_Alarmes[1, 58].Active := GVL_RegTROX.RegSouf_PD_FCVT02_DefCom;

//Alarme 59
GA_Alarmes[1, 59].Id := 59;
GA_Alarmes[1, 59].Libelle := 'Défaut discordance débit du Registre de soufflage petit débit';
GA_Alarmes[2, 59].Libelle := 'Mismatch Flow Rate of Low-flow blow damper';
GA_Alarmes[1, 59].Active := GVL_RegTROX.RegSouf_PD_FCVT02_Def_DiscordDeb;

//Alarme 60
GA_Alarmes[1, 60].Id := 60;
GA_Alarmes[1, 60].Libelle := 'Défaut communication du Registre de soufflage général';
GA_Alarmes[2, 60].Libelle := 'General blow damper communication fault';
GA_Alarmes[1, 60].Active := GVL_RegTROX.RegSouf_Cabine_FCVT03_DefCom;

//Alarme 61
GA_Alarmes[1, 61].Id := 61;
GA_Alarmes[1, 61].Libelle := 'Défaut discordance débit du Registre de soufflage général';
GA_Alarmes[2, 61].Libelle := 'Mismatch Flow Rate of General blow damper';
GA_Alarmes[1, 61].Active := GVL_RegTROX.RegSouf_Cabine_FCVT03_Def_DiscordDeb;

//Alarme 62
GA_Alarmes[1, 62].Id := 62;
GA_Alarmes[1, 62].Libelle := 'Défaut communication du Registre de bypass de la CTA climatique';
GA_Alarmes[2, 62].Libelle := 'Climatic AHU bypass damper communication fault';
GA_Alarmes[1, 62].Active := GVL_RegTROX.Reg_Bypass_FCVT04_DefCom;

//Alarme 63
GA_Alarmes[1, 63].Id := 63;
GA_Alarmes[1, 63].Libelle := 'Défaut discordance débit du Registre de bypass de la CTA climatique';
GA_Alarmes[2, 63].Libelle := 'Mismatch Flow Rate of Climatic AHU bypass damper';
GA_Alarmes[1, 63].Active := GVL_RegTROX.Reg_Bypass_FCVT04_Def_DiscordDeb;

//Alarme 64
GA_Alarmes[1, 64].Id := 64;
GA_Alarmes[1, 64].Libelle := 'Défaut communication du Registre de soufflage gros débit de la cabine';
GA_Alarmes[2, 64].Libelle := 'High-flow booth blower damper communication fault';
GA_Alarmes[1, 64].Active := GVL_RegTROX.RegSouf_CabGD_FCVT05_DefCom;

//Alarme 65
GA_Alarmes[1, 65].Id := 65;
GA_Alarmes[1, 65].Libelle := 'Défaut discordance débit du Registre de soufflage gros débit de la cabine';
GA_Alarmes[2, 65].Libelle := 'Mismatch Flow Rate of High-flow booth blower damper';
GA_Alarmes[1, 65].Active := GVL_RegTROX.RegSouf_CabGD_FCVT05_Def_DiscordDeb;

//Alarme 66
GA_Alarmes[1, 66].Id := 66;
GA_Alarmes[1, 66].Libelle := 'Défaut communication du Registre de soufflage petit débit de la cabine';
GA_Alarmes[2, 66].Libelle := 'Booth low-flow blow damper communication fault';
GA_Alarmes[1, 66].Active := GVL_RegTROX.RegSouf_CabPD_FCVT06_DefCom;

//Alarme 67
GA_Alarmes[1, 67].Id := 67;
GA_Alarmes[1, 67].Libelle := 'Défaut discordance débit du Registre de soufflage petit débit de la cabine';
GA_Alarmes[2, 67].Libelle := 'Mismatch Flow Rate of Booth low-flow blow damper';
GA_Alarmes[1, 67].Active := GVL_RegTROX.RegSouf_CabPD_FCVT06_Def_DiscordDeb;

//Alarme 68
GA_Alarmes[1, 68].Id := 68;
GA_Alarmes[1, 68].Libelle := 'Défaut communication du Registre de reprise de la CTA climatique';
GA_Alarmes[2, 68].Libelle := 'Climatic AHU recovery damper communication fault';
GA_Alarmes[1, 68].Active := GVL_RegTROX.RegRep_FCVT07_DefCom;

//Alarme 69
GA_Alarmes[1, 69].Id := 69;
GA_Alarmes[1, 69].Libelle := 'Défaut discordance débit du Registre de reprise de la CTA climatique';
GA_Alarmes[2, 69].Libelle := 'Mismatch Flow Rate of Climatic AHU recovery damper';
GA_Alarmes[1, 69].Active := GVL_RegTROX.RegRep_FCVT07_Def_DiscordDeb;

// idx = compteur d'alarmes actives
idx := 0;

// Parcours de toutes les alarmes (on utilise la langue 1 comme référence logique)
FOR i := 1 TO NB_ALARMES_MAX DO

    // On teste seulement la version FR pour la logique (Id + Active)
    IF GA_Alarmes[1, i].Id <> 0 THEN

        IF GA_Alarmes[1, i].Active THEN
            idx := idx + 1;

            // On recopie les deux langues dans le tableau "actives"
            // 1 = FR, 2 = EN
            GA_AlarmesActives[1, idx] := GA_Alarmes[1, i];
            GA_AlarmesActives[2, idx] := GA_Alarmes[2, i];
        END_IF

    END_IF

END_FOR

// Nettoyage des cases non utilisées pour les deux langues
FOR i := idx + 1 TO NB_ALARMES_MAX DO
    // FR
    GA_AlarmesActives[1, i].Id      := 0;
    GA_AlarmesActives[1, i].Libelle := '';
    GA_AlarmesActives[1, i].Active  := FALSE;

    // EN
    GA_AlarmesActives[2, i].Id      := 0;
    GA_AlarmesActives[2, i].Libelle := '';
    GA_AlarmesActives[2, i].Active  := FALSE;
END_FOR

// Mise à jour du compteur
G_NbAlarmesActives := idx;

// ------------------------------------------------------------
// COPIE DES LIBELLÉS DANS Tab_Alarme_FREN (FR + EN uniquement)
// ------------------------------------------------------------
FOR i := 1 TO G_NbAlarmesActives DO
    Tab_Alarme_FREN[1, i] := GA_AlarmesActives[1, i].Libelle;   // Français
    Tab_Alarme_FREN[2, i] := GA_AlarmesActives[2, i].Libelle;   // Anglais
END_FOR

// Nettoyage des lignes restantes jusqu'à 100
FOR i := G_NbAlarmesActives + 1 TO 100 DO
    Tab_Alarme_FREN[1, i] := '';
    Tab_Alarme_FREN[2, i] := '';
END_FOR

//Variable des alarmes warning
Mode_Warning := Defaut_Porte_Ouverte OR Defaut_Com_Dalcnet OR Defaut_Com_Vanne_General OR Defaut_Com_Vanne_General
			OR Defaut_Com_Client OR Defaut_Discord_Deb_Ext OR Defaut_Discord_Deb_Souf OR Defaut_Discord_Reg_Ext_Ferm
			OR Defaut_Discord_Reg_Souf_Ferm OR Defaut_Klixon_BattElec OR Defaut_Discord_Regul_Press_Cab
			OR Defaut_Com_Reg_Souf OR Defaut_Com_Reg_Ext OR Defaut_Ensemble_Bas_Debit OR Defaut_Ensemble_Bypass
			OR Defaut_Sonde_Press_Cabine OR Defaut_Sonde_Temp_Cabine OR Defaut_Sonde_Hygro_Cabine
			OR Defaut_Sonde_Temp_Eau_Mitig OR Defaut_Hygrostat_CTA OR Defaut_Regul_Temp OR Defaut_Regul_Hygro
			OR Defaut_Discord_Souf_CTA
			OR GVL_RegTROX.RegSouf_GD_FCVT01_DefCom	OR GVL_RegTROX.RegSouf_GD_FCVT01_Def_DiscordDeb	OR GVL_RegTROX.RegSouf_PD_FCVT02_DefCom
			OR GVL_RegTROX.RegSouf_PD_FCVT02_Def_DiscordDeb	OR GVL_RegTROX.RegSouf_Cabine_FCVT03_DefCom	 OR GVL_RegTROX.RegSouf_Cabine_FCVT03_Def_DiscordDeb
			OR GVL_RegTROX.Reg_Bypass_FCVT04_DefCom OR GVL_RegTROX.Reg_Bypass_FCVT04_Def_DiscordDeb OR GVL_RegTROX.RegSouf_CabGD_FCVT05_DefCom
			OR GVL_RegTROX.RegSouf_CabGD_FCVT05_Def_DiscordDeb OR GVL_RegTROX.RegSouf_CabPD_FCVT06_DefCom OR GVL_RegTROX.RegSouf_CabPD_FCVT06_Def_DiscordDeb
			OR GVL_RegTROX.RegRep_FCVT07_DefCom OR GVL_RegTROX.RegRep_FCVT07_Def_DiscordDeb;

END_PROGRAM

// ---- POUs/Block/Cabines/Humidificateur.TcPOU
FUNCTION_BLOCK Humidificateur
VAR_INPUT
	Enable				:BOOL;
	Cmd_Humidificateur	:BOOL;
	Cons_Humi_Dem		:REAL;	(*Consigne humidificateur demandé (venant de la Régulation) / en %*)
	Info_Defaut			:BOOL;	(*VAR_INPUT	Info défaut hygrostat/ 1 = Défaut*)
	Inverse_SAN			:BOOL;	(*Inversion de la sortie SAN / 1 = Sens inverse / 0 = Sens normal*)
	SAN_OUT_MIN			:REAL;	(*Valeur minimal de la sortie SAN / en point automate*)
	SAN_OUT_MAX			:REAL;	(*Valeur maximal de la sortie SAN / en point automate*)
END_VAR

VAR_OUTPUT
	SAN_CONS_HUMI	:INT;	(*Consigne a appliqué (pour SAN) / en %*)
	STOR_CMD_HUMI	:BOOL;	(*VAR_OUTPUT	Commande a appliqué / 1 = Marche*)
END_VAR

VAR
	val_x				:REAL;
	val_b				:REAL;
	val_a				:REAL;
	val_y				:REAL;
	val_final				:REAL;
END_VAR

(* Gestion consigne **************************************************************)
IF (Enable AND NOT Info_Defaut)
	THEN (* Gestion sortie analogique *)
		(* Mise à l'echelle sortie ****)
		val_x := Cons_Humi_Dem;
		val_b := SAN_OUT_MAX - (val_a * 100.0);
		val_a := (SAN_OUT_MAX - SAN_OUT_MIN) / 100.0;
		val_y := (val_a * val_x) + val_b;

		(* Inversion de la sortie ANA ****)
		IF (Inverse_SAN)
			THEN
				val_final := SAN_OUT_MAX - val_y;
			ELSE
				val_final := val_y;
		END_IF;
		SAN_CONS_HUMI := REAL_TO_INT(LIMIT(SAN_OUT_MIN,val_final, SAN_OUT_MAX));
		STOR_CMD_HUMI := Cmd_Humidificateur;
	ELSE (* Gestion sortie TOR PWM *)
		SAN_CONS_HUMI := 0;
		STOR_CMD_HUMI := FALSE;
END_IF;

END_FUNCTION_BLOCK

// ---- POUs/Gestion_Enceinte_Clim/B_Gestion_Defaut.TcPOU
PROGRAM B_Gestion_Defaut
VAR
(*Alarme défaut régulation de température*)
	TON_Ecart_Temp: TON;
(*Alarme défaut régulation d'hygrométrie*)
	TON_Ecart_Hygro: TON;
(*Alarme défaut de discordance de soufflage entre le pressostat de sécurité et les moteurs de la CTA*)
	TON_Defaut_Discord_Souf: TON;
(*Alarme défaut du thermostat de sécurité automatique proche de la batterie électrique*)
	RS_Thermostat_Secu: RS;
	TON_1: TON;
END_VAR

(**********************************************Alarme défaut moteur 1 de soufflage CTA*)
Defaut_MotRep_CTA := NOT E_Def_MotRep_CTA;

(**********************************************Alarme défaut moteur 2 de soufflage CTA*)
Defaut_MotSouf_CTA := NOT E_Def_MotSouf_CTA;

(**********************************************Alarme défaut hygrostat de soufflage*)
Defaut_Hygrostat_CTA := NOT E_Hygrostat_Souf_CTA;

(**********************************************Alarme défaut sur l'alimentation électrique de la batterie électrique*)
Defaut_Alim_BatElec_CTA := NOT E_Def_Alim_BatElec_CTA;

(**********************************************Alarme défaut sur l'humidificateur*)
Defaut_Humi_CTA := NOT E_Def_Humi_CTA;

(**********************************************Alarme défaut régulation de température*)
TON_Ecart_Temp(IN:= ((S_Ecart_Regul_PID_Temp > TOL_Regul_Temp_EnceintClim) AND Mode_Cabine_Automatique) , PT:= t#100m );
IF(TON_Ecart_Temp.Q)
	THEN
	Defaut_Regul_Temp := TRUE;
	ELSE
	Defaut_Regul_Temp := FALSE;
END_IF;

(**********************************************Alarme défaut régulation d'hygrométrie*)
TON_Ecart_Hygro(IN:= ((S_Ecart_Regul_PID_Hygro > TOL_Regul_Hygro_EnceintClim) AND Mode_Cabine_Automatique) , PT:= t#100m );
IF(TON_Ecart_Hygro.Q)
	THEN
	Defaut_Regul_Hygro := TRUE;
	ELSE
	Defaut_Regul_Hygro := FALSE;
END_IF;

(*Defaut generale sur la partie humidification*)
Defaut_General_Humi := Defaut_Sonde_Hygro_Cabine OR Defaut_Humi_CTA;

(*Defaut des défauts qui arrêtent la recette du mode 25*)
Defaut_Arret_Mode25 := 	Defaut_MotRep_CTA OR Defaut_MotSouf_CTA
						 OR Defaut_Alim_BatElec_CTA OR Defaut_Humi_CTA
						OR Defaut_Sonde_Hygro_Cabine OR Defaut_Sonde_Temp_Cabine
						OR Defaut_Thermostat_Secu OR Defaut_Sonde_Temp_Souf;
						
(**********************************************Alarme défaut de discordance de soufflage entre le pressostat de sécurité et les moteurs de la CTA*)
TON_Defaut_Discord_Souf(IN:= NOT E_Pressostat_Secu AND (Cons_Actionneur_Mot1_Souf_CTA > 60) AND (Cons_Actionneur_Mot2_Souf_CTA > 60), PT:= T#60S);
IF (TON_Defaut_Discord_Souf.Q)
	THEN
	Defaut_Discord_Souf_CTA	:= TRUE;
	ELSE
	Defaut_Discord_Souf_CTA	:= FALSE;	
END_IF

(**********************************************Alarme défaut du thermostat de sécurité automatique proche de la batterie électrique*)
TON_1(IN:= NOT E_Thermostat_Secu  , PT:= T#1S );
RS_Thermostat_Secu(SET:= TON_1.Q, RESET1:= Cmd_Rearmement, Q1=> Defaut_Thermostat_Secu);

END_PROGRAM

// ---- POUs/Gestion_Enceinte_Clim/C0_Gestion_Consignes.TcPOU
PROGRAM C0_Gestion_Consignes
VAR
(*Gestion du post ventilation*)
	TON_Post_Ventilation: TON;
	Temp_Post_ventil: TIME;
	RS_Post_ventilation: RS;
	Reset_Post_Ventil: BOOL;
	R_Trig_Post_Ventil: R_TRIG;
	TP_Post_Ventil: TP;
	Arret_Post_Ventil: BOOL;
	Set_Post_Ventilation: BOOL;
	Set_TON: BOOL;
	RS_YMin: RS;
	TP_YMin: TP;
	Var_1: BOOL;
	TON_YMin: TON;
	R_TRIG_TempHygro: R_TRIG;
END_VAR

(**********************************************Gestion des consignes lors du Mode Stand-By (Libre)
IF(Mode_Cabine_Libre)
	THEN
	Lect_Cons_Temperature_Cabine		:= 0.0 ;
	Lect_Cons_Hygrometrie_Cabine			:= 0.0 ;
	Lect_Cons_VitMot_Cabine_MEnCond		:= 0.0 ;
END_IF;*)

(**********************************************Gestion des consignes lors du Mode Mise en fonctionnement*)
Mode_MEnCond := Mode_Auto.Mode_25;
Mode_Fctnmt := Mode_Auto.Mode_28;
(*Maintient de la consigne de température et de l'hygrométrie durant toute la recette si il y'a eu un mode mise en condition*)
RS_MEnCond(SET:= (Mode_Cabine_Automatique AND Mode_MEnCond), RESET1:= Mode_Cabine_Libre  OR (Numero_Mode_Actuel = 10));
IF(RS_MEnCond.Q1)
	THEN
	(*Gestion du changement de vitesse des moteurs de la CTA une fois la mise en condition terminée*)
	IF(Mode_MEnCond)
		THEN
		Lect_Cons_VitMot_Cabine_MEnCond		:= Cons_VitMot_Cabine_MEnCond;
		ELSE
		Lect_Cons_VitMot_Cabine_MEnCond		:= Cons_VitMot_Cabine_EnCond;
	END_IF;
	ELSE
	Lect_Cons_VitMot_Cabine_MEnCond := 0.0;
END_IF;
(*Enregistrement des consignes sur le front montant du mode qui gére les consigne (Mode 25)*)
R_TRIG_TempHygro(CLK:= Mode_MEnCond);
IF (R_TRIG_TempHygro.Q)
	THEN
	Lect_Cons_Temperature_Cabine			:= Mode_Auto.Out_Para_11;
	Lect_Cons_Hygrometrie_Cabine			:= Mode_Auto.Out_Para_12;
	ELSE
	Lect_Cons_Temperature_Cabine			:= Lect_Cons_Temperature_Cabine;
	Lect_Cons_Hygrometrie_Cabine			:= Lect_Cons_Hygrometrie_Cabine;
END_IF

(**********************************************Gestion de l'enable PID de la température*)
IF(RS_MEnCond.Q1 AND NOT Defaut_Sonde_Temp_Cabine AND NOT Defaut_Alim_BatElec_CTA AND E_Pressostat_Secu)
	THEN
	Enable_Regul_PID_Temp := TRUE AND NOT Dmd_Post_Ventilation;
	ELSE
	Enable_Regul_PID_Temp := FALSE;
END_IF;

(**********************************************Gestion de l'enable PID de l'hygrometrie*)
IF(RS_MEnCond.Q1  AND NOT Defaut_General_Humi AND E_Pressostat_Secu)
	THEN
	Enable_Regul_PID_Hr := TRUE AND NOT Dmd_Post_Ventilation;
	ELSE
	Enable_Regul_PID_Hr := FALSE;
END_IF;
(*Passage à la consigne minimum à 18% de l'humidification, si demande*)
Var_1 := (S_Cmd_Regul_PID_Humi >= 7.0);
TON_YMin(IN:= Var_1, PT:= T#30s);
RS_YMin(SET:= (Enable_Regul_PID_Humi AND TON_YMin.Q), RESET1:= (Mode_Arret_Auto OR (Numero_Mode_Actuel = 10)));
TP_YMin(IN:= RS_YMin.Q1, PT:= T#1s);
IF (TP_YMin.Q) THEN Regul_Humi_YMin := 25.0; ELSE Regul_Humi_YMin := 0.0; END_IF;

(**********************************************Gestion du post ventilation*)
(*Conversion du temp - temps en seconde*)
Temp_Post_ventil 		:= TO_TIME((TO_DINT(Cons_Sec_Post_Ventil + 5)) * 1000);
(*Détection de la chauffe*)
Set_Post_Ventilation 	:= (S_Cmd_Regul_PID_Temp_Chaud > 10.0);
Set_TON 				:= (S_Cmd_Regul_PID_Temp_Chaud < 10.0);
TON_Post_Ventilation	(IN:= (Set_TON), PT:= Temp_Post_ventil);
RS_Post_ventilation		(SET:= Set_Post_Ventilation,
						RESET1:= Reset_Post_Ventil OR Numero_Mode_Auto=0);
Reset_Post_Ventil 		:= TON_Post_Ventilation.Q AND NOT TP_Post_Ventil.Q;
(*Détection d'un arrêt lors du front montant de l'arrêt de la recette*)
Arret_Post_Ventil 		:= (Mode_Arret_Auto (*OR (Numero_Mode_Actuel = 10)*));
R_Trig_Post_Ventil		(CLK:= Arret_Post_Ventil);
TP_Post_Ventil			(IN:= R_Trig_Post_Ventil.Q, PT:= Temp_Post_ventil);
(*Mode post ventilation*)
Dmd_Post_Ventilation 	:= TP_Post_Ventil.Q AND RS_Post_ventilation.Q1;

END_PROGRAM

// ---- POUs/Gestion_Enceinte_Clim/C_Regul_Temp.TcPOU
PROGRAM C_Regul_Temp
VAR
	TON_Chaud: TON;
	TON_Froid: TON;
	Cons_Regul_Chaud: REAL;
	Cons_Regul_Froid: REAL;
	Interdiction_Chaud: BOOL;
	Interdiction_Froid: BOOL;
	Bool_Reg_chaud: BOOL;
	Bool_Reg_froid: BOOL;
	Grad_Cons: UP_DOWN_RATE;
	Calc_Cons_Chaud: REAL;
	Regul_Souf_Chaud: PID;
	Inter_Souf_Chaud: BOOL;
	Regul_Temp_Chaud: OSCAT_BASIC.CTRL_PID;
	Sup_PID_Cd: REAL := 0;
	Regul_Temp_Froid: OSCAT_BASIC.CTRL_PID;
	Sup_PID_Fd: REAL := 0;
	Ecart_TempPiece_Consigne: REAL;
	TOF_Stop: TOF;
	RS_enable: RS;
	Regul_Temp_Amb: OSCAT_BASIC.CTRL_PID;
	Consigne_Soufflage: REAL;
END_VAR
VAR // added by the converter: edge detectors and wires of the graphical bodies
    _w1 : REAL;
    _w2, _w3, _w4 : ANY;
END_VAR

Consigne_Soufflage := _w1;
RS_enable(SET := Tab_MES_Sonde_Temp_Amb.R_MesCor > Lect_Cons_Temperature_Cabine + 2.0, RESET1 := Tab_MES_Sonde_Temp_Amb.R_MesCor < Lect_Cons_Temperature_Cabine - 2.0); // RS
Enable_Regul_PID_Temp_Chaud := _w2;
_w2 := Enable_Regul_PID_Temp AND NOT RS_enable.Q1;
Enable_Regul_PID_Temp_Froid := Enable_Regul_PID_Temp AND RS_enable.Q1;
// Gestion passage PID chaud/Froid
Cons_Regul_Froid := Consigne_Soufflage + Offset_Regul_PID_Temp;
Cons_Regul_Chaud := Consigne_Soufflage - Offset_Regul_PID_Temp;
_w1 := LIMIT(Limit_Min_Souf, Regul_Temp_Amb.Y + Lect_Cons_Temperature_Cabine, Limit_Max_Souf);
TON_Chaud(IN := Tab_MES_Sonde_Temp_Amb.R_MesCor < Cons_Regul_Chaud, PT := T#30s); // TON
// Boucle de régulation
Regul_Temp_Amb(
    ACT := Tab_MES_Sonde_Temp_Amb.R_MesCor,
    SET := Lect_Cons_Temperature_Cabine,
    SUP := 0.0,
    OFS := 0.0,
    M_I := 0.0,
    MAN := NOT Enable_Regul_PID_Temp,
    RST := NOT Enable_Regul_PID_Temp,
    KP := Kp_Ambiance,
    TN := Ki_Ambiance,
    TV := Kd_Ambiance,
    LL := -11.0,
    LH := 11.0); // OSCAT_BASIC.CTRL_PID
Interdiction_Froid := Enable_Regul_PID_Temp_Chaud AND TON_Chaud.Q;
TON_Froid(IN := Tab_MES_Sonde_Temp_Amb.R_MesCor > Cons_Regul_Froid, PT := T#30s); // TON
Interdiction_Chaud := Enable_Regul_PID_Temp_Froid AND TON_Froid.Q;
Grad_Cons(
    IN_CONS := SEL(Enable_Regul_PID_Temp_Chaud, Tab_MES_Sonde_Temp_Amb.R_MesCor, Cons_Regul_Chaud),
    IN_UP_RATE := 1.0,
    IN_DOWN_RATE := 1.0,
    TIME_STEP := T#30s,
    MODE := 2); // UP_DOWN_RATE
Calc_Cons_Chaud := Grad_Cons.OUT_CONS;
TOF_Stop(IN := Tab_Mes_Sonde_Temp_Souf.R_MesCor > 50, PT := T#2m); // TOF
Inter_Souf_Chaud := TOF_Stop.Q;
Regul_Temp_Chaud(
    ACT := Tab_Mes_Sonde_Temp_Souf.R_MesCor,
    SET := Cons_Regul_Chaud,
    SUP := Sup_PID_Cd,
    OFS := 0.0,
    M_I := 0.0,
    MAN := NOT Enable_Regul_PID_Temp_Chaud,
    RST := NOT Enable_Regul_PID_Temp_Chaud,
    KP := Gain_Regul_PID_Temp_Chaud,
    TN := Integral_Regul_PID_Temp_Chaud,
    TV := Derive_Regul_PID_Temp_Chaud,
    LL := 0.0,
    LH := Cons_Maxi_Bat_Electrique); // OSCAT_BASIC.CTRL_PID
S_Cmd_Regul_PID_Temp_Chaud := SEL(Inter_Souf_Chaud, Regul_Temp_Chaud.Y, 0.0);
Bool_Reg_chaud := Regul_Temp_Chaud.Y > 5.0;
Regul_Temp_Froid(
    ACT := Tab_Mes_Sonde_Temp_Souf.R_MesCor,
    SET := Cons_Regul_Froid,
    SUP := Sup_PID_Fd,
    OFS := 0.0,
    M_I := 0.0,
    MAN := NOT Enable_Regul_PID_Temp_Froid,
    RST := NOT Enable_Regul_PID_Temp_Froid,
    KP := Gain_Regul_PID_Temp_Froid,
    TN := Integral_Regul_PID_Temp_Froid,
    TV := Derive_Regul_PID_Temp_Froid,
    LL := -100.0,
    LH := 0.0); // OSCAT_BASIC.CTRL_PID
_w3 := ABS(Regul_Temp_Froid.Y);
S_Cmd_Regul_PID_Temp_Froid := SEL(FALSE, _w3, 0.0);
Bool_Reg_froid := _w3 > 5.0;
// Gestion discordance
_w4 := Lect_Cons_Temperature_Cabine - Tab_MES_Sonde_Temp_Amb.R_MesCor;
Ecart_TempPiece_Consigne := _w4;
S_Ecart_Regul_PID_Temp := SEL(Enable_Regul_PID_Temp, 0.0, ABS(_w4));

END_PROGRAM

// ---- POUs/Block/Autres/UP_DOWN_RATE.TcPOU
FUNCTION_BLOCK UP_DOWN_RATE
VAR_INPUT
    IN_CONS      : REAL;    // Consigne cible à atteindre
    IN_UP_RATE   : REAL;    // Pas d'incrémentation (valeur ajoutée à chaque pas)
    IN_DOWN_RATE : REAL;    // Pas de décrémentation (valeur retirée à chaque pas)
    TIME_STEP    : TIME;    // Intervalle entre chaque évolution (ex : T#1s)
    MODE         : INT;     // Mode de fonctionnement : 0 = UP+DOWN, 1 = DOWN seulement, 2 = UP seulement
END_VAR

VAR_OUTPUT
    OUT_CONS     : REAL;    // Valeur évolutive vers la consigne
END_VAR

VAR
    ton_step     : TON;     // Temporisateur cyclique pour le pas de temps
    r_trig_step  : R_TRIG;  // Détecteur de front montant du temporisateur
END_VAR

// --- Temporisateur cyclique ---
ton_step(IN := NOT ton_step.Q, PT := TIME_STEP);

// --- Détection du front montant du timer ---
r_trig_step(CLK := ton_step.Q);

// --- Collage instantané si besoin ---
CASE MODE OF
    2: // --- Mode UP uniquement ---
        IF OUT_CONS > IN_CONS THEN
            OUT_CONS := IN_CONS;   // Collage immédiat si consigne descend d’un coup
        END_IF
    1: // --- Mode DOWN uniquement ---
        IF OUT_CONS < IN_CONS THEN
            OUT_CONS := IN_CONS;   // Collage immédiat si consigne monte d’un coup
        END_IF
END_CASE

// --- Mise à jour de la sortie uniquement au front montant du timer ---
IF r_trig_step.Q THEN
    CASE MODE OF
        0: // --- Mode UP+DOWN (les deux directions) ---
            IF OUT_CONS < IN_CONS THEN
                OUT_CONS := OUT_CONS + IN_UP_RATE;         // On incrémente
                IF OUT_CONS > IN_CONS THEN
                    OUT_CONS := IN_CONS;                   // On ne dépasse jamais la consigne
                END_IF
            ELSIF OUT_CONS > IN_CONS THEN
                OUT_CONS := OUT_CONS - IN_DOWN_RATE;       // On décrémente
                IF OUT_CONS < IN_CONS THEN
                    OUT_CONS := IN_CONS;
                END_IF
            END_IF
        1: // --- Mode DOWN uniquement ---
            IF OUT_CONS > IN_CONS THEN
                OUT_CONS := OUT_CONS - IN_DOWN_RATE;       // On décrémente seulement
                IF OUT_CONS < IN_CONS THEN
                    OUT_CONS := IN_CONS;
                END_IF
            END_IF
        2: // --- Mode UP uniquement ---
            IF OUT_CONS < IN_CONS THEN
                OUT_CONS := OUT_CONS + IN_UP_RATE;         // On incrémente seulement
                IF OUT_CONS > IN_CONS THEN
                    OUT_CONS := IN_CONS;
                END_IF
            END_IF
    END_CASE
END_IF

END_FUNCTION_BLOCK

// ---- POUs/Gestion_Enceinte_Clim/D_Regul_Humi.TcPOU
PROGRAM D_Regul_Humi
VAR
	TON_Humi: TON;
	TOF_Deshu: TOF;

	Cons_Regul_Humi: REAL;
	Cons_Regul_Deshu: REAL;
	Interdiction_Humi: BOOL;
	Interdiction_Deshu: BOOL;
	Bool_Reg_Humi: BOOL;
	Bool_Reg_Deshu: BOOL;
	
	Regul_humidification: OSCAT_BASIC.CTRL_PID;
	Sup_PID_humi: REAL := 0;
	Regul_Deshumidification: OSCAT_BASIC.CTRL_PID;
	Sup_PID_Deshu: REAL := 0;
	SCL_Real_Humi: SCL_Real;
	SCL_Real_Deshu: SCL_Real;
	Dew_Point_Mes: Dew_Point;
	Dew_Point_Cons: Dew_Point;
	Mesure_Dew_Point: REAL;
	Consigne_Dew_Point: REAL;
	RS_Deshu: RS;
	RS_enable: RS;
END_VAR
VAR // added by the converter: edge detectors and wires of the graphical bodies
    _w1, _w3, _w4 : ANY;
    _w2 : BOOL;
END_VAR

RS_enable(SET := Tab_MES_Sonde_Hygro_Amb.R_MesCor > Lect_Cons_Hygrometrie_Cabine + 5.0, RESET1 := _w1); // RS
_w3 := Enable_Regul_PID_Hr AND _w2;
// Gestion passage PID humidification/deshumidification
Cons_Regul_Deshu := Lect_Cons_Hygrometrie_Cabine + Offset_Regul_PID_Hr;
_w1 := Tab_MES_Sonde_Hygro_Amb.R_MesCor < Lect_Cons_Hygrometrie_Cabine - 5.0;
_w2 := NOT RS_enable.Q1;
Cons_Regul_Humi := Lect_Cons_Hygrometrie_Cabine - Offset_Regul_PID_Hr;
Enable_Regul_PID_Humi := _w3;
Enable_Regul_PID_Deshu := Enable_Regul_PID_Hr AND RS_enable.Q1;
TON_Humi(IN := Tab_MES_Sonde_Hygro_Amb.R_MesCor < Lect_Cons_Hygrometrie_Cabine - 3.0, PT := T#10s); // TON
Interdiction_Deshu := Enable_Regul_PID_Humi AND TON_Humi.Q;
RS_Deshu(SET := Tab_MES_Sonde_Hygro_Amb.R_MesCor > Lect_Cons_Hygrometrie_Cabine + 10.0, RESET1 := Tab_MES_Sonde_Hygro_Amb.R_MesCor < Lect_Cons_Hygrometrie_Cabine); // RS
Interdiction_Humi := RS_Deshu.Q1 AND Enable_Regul_PID_Deshu;
// Calcul du point de rosé
Dew_Point_Mes(rTemp := Tab_MES_Sonde_Temp_Amb.R_MesCor, rRh := Tab_MES_Sonde_Hygro_Amb.R_MesCor); // Dew_Point
Mesure_Dew_Point := Dew_Point_Mes.rDewPoint;
Dew_Point_Cons(rTemp := Lect_Cons_Temperature_Cabine, rRh := Lect_Cons_Hygrometrie_Cabine); // Dew_Point
Consigne_Dew_Point := Dew_Point_Cons.rDewPoint;
// Boucle de régulation
Regul_humidification(
    ACT := Tab_MES_Sonde_Hygro_Amb.R_MesCor,
    SET := Cons_Regul_Humi,
    SUP := Sup_PID_humi,
    OFS := 0.0,
    M_I := 0.0,
    MAN := NOT Enable_Regul_PID_Humi,
    RST := NOT Enable_Regul_PID_Humi,
    KP := Gain_Regul_PID_Humi,
    TN := Integral_Regul_PID_Humi,
    TV := Derive_Regul_PID_Humi,
    LL := 0.0,
    LH := Cons_Maxi_Humidificateur); // OSCAT_BASIC.CTRL_PID
S_Cmd_Regul_PID_Humi := SEL(Interdiction_Humi, Regul_humidification.Y, 0.0);
Bool_Reg_Humi := Regul_humidification.Y > 5.0;
Regul_Deshumidification(
    ACT := Tab_MES_Sonde_Hygro_Amb.R_MesCor,
    SET := Cons_Regul_Deshu,
    SUP := Sup_PID_Deshu,
    OFS := 0.0,
    M_I := 0.0,
    MAN := NOT Enable_Regul_PID_Deshu,
    RST := NOT Enable_Regul_PID_Deshu,
    KP := Gain_Regul_PID_Deshu,
    TN := Integral_Regul_PID_Deshu,
    TV := Derive_Regul_PID_Deshu,
    LL := -100.0,
    LH := 0.0); // OSCAT_BASIC.CTRL_PID
_w4 := ABS(Regul_Deshumidification.Y);
S_Cmd_Regul_PID_Deshu := SEL(FALSE, _w4, 0.0);
Bool_Reg_Deshu := _w4 > 5.0;
// Gestion discordance
S_Ecart_Regul_PID_Hygro := SEL(Enable_Regul_PID_Hr, 0.0, ABS(Tab_MES_Sonde_Hygro_Amb.R_MesCor - Lect_Cons_Hygrometrie_Cabine));

END_PROGRAM

// ---- POUs/Block/Autres/SCL_Real.TcPOU
FUNCTION_BLOCK SCL_Real
VAR_INPUT
	IN_REAL: REAL;
	LIM_MIN_IN_REAL: REAL;
	LIM_MAX_IN_REAL: REAL;
	LIM_MIN_OUT_REAL: REAL;
	LIM_MAX_OUT_REAL: REAL;
END_VAR
VAR_OUTPUT
	OUT_REAL: REAL;
END_VAR
VAR
	val_final: REAL;
	TON_1: TON;
	SCL_OUT: REAL;
	TON_2: TON;
	val_b: REAL;
	val_a: REAL;
	val_y: REAL;
	val_x: REAL;
	LIM_MAX_IN: REAL;
	LIM_MAX_OUT: REAL;
	SCL_IN: REAL;
END_VAR

(* Sécurité anti division / 0 *)

TON_1(IN := TRUE, PT := t#1s);
LIM_MAX_IN := SEL(TON_1.Q, 1.0, LIM_MAX_IN_REAL);

IF ((LIM_MAX_IN - LIM_MIN_IN_REAL) = 0.0)
	THEN
		SCL_IN := 1.0;
	ELSE
		SCL_IN := LIM_MAX_IN - LIM_MIN_IN_REAL;
END_IF;

TON_2(IN := TRUE, PT := t#1s);
LIM_MAX_OUT := SEL(TON_2.Q, 1.0, LIM_MAX_OUT_REAL);

IF ((LIM_MAX_OUT - LIM_MIN_OUT_REAL) = 0.0)
	THEN
		SCL_OUT := 1.0;
	ELSE
		SCL_OUT := LIM_MAX_OUT - LIM_MIN_OUT_REAL;
END_IF;

(* Mise à l'échelle *)

val_x := IN_REAL;

val_b := LIM_MAX_OUT_REAL - (val_a * LIM_MAX_IN_REAL);

val_a := (SCL_OUT) / MAX(0.1,(SCL_IN));

val_y := (val_a * val_x) + val_b;


(* Traitement final *)

val_final := val_y;
OUT_REAL := LIMIT(0.0, val_final, 100.0);

(*Sécurité valeur maximum d'entrée à zéro
IF (LIM_MAX_IN_REAL = 0)
	THEN
	OUT_REAL := 0.0;
END_IF;*)

END_FUNCTION_BLOCK

// ---- POUs/Block/Autres/Dew_Point.TcPOU
FUNCTION_BLOCK Dew_Point
VAR_INPUT
    rTemp : REAL; (* Température ambiante [°C] *)
    rRh   : REAL; (* Humidité Relative [%] *)
END_VAR
VAR_OUTPUT
    rDewPoint : REAL; (* Point de rosée calculé [°C] *)
    bError    : BOOL; (* TRUE si les entrées sont incohérentes (ex: sonde HS) *)
END_VAR
VAR
    rGamma   : REAL;
    rRh_Safe : REAL; (* Valeur interne sécurisée pour le calcul *)
    
    (* Constantes Magnus-Tetens *)
    c_b : REAL := 17.62;
    c_c : REAL := 243.12;
END_VAR

(* 1. Gestion des erreurs et sécurisation *)
bError := (rRh < 0.0) OR (rRh > 100.0) OR (rTemp < -19.0);

(* On borne l'humidité pour protéger le Logarithme (LN) *)
(* Même si le capteur envoie -10% (rupture de fil), on calcule avec 0.1% pour éviter le crash PLC *)
IF rRh < 0.1 THEN
    rRh_Safe := 0.1; 
ELSIF rRh > 100.0 THEN
    rRh_Safe := 100.0;
ELSE
    rRh_Safe := rRh;
END_IF

(* 2. Calcul du coefficient Gamma *)
(* Formule : ln(RH/100) + (b * T) / (c + T) *)
rGamma := LN(rRh_Safe / 100.0) + ( (c_b * rTemp) / (c_c + rTemp) );

(* 3. Résultat final *)
rDewPoint := (c_c * rGamma) / (c_b - rGamma);

END_FUNCTION_BLOCK

// ---- POUs/Gestion_Enceinte_Clim/E_Cons_Cmd_Actionneurs.TcPOU
PROGRAM E_Cons_Cmd_Actionneurs
VAR
	Calcul1: REAL;
	mini_humi: REAL;
	SCL_Real_Decal_Deshu: SCL_Real;
END_VAR

(**********************************************Gestion de la vanne 3 voies de régulation*)
Calcul1 := S_Cmd_Regul_PID_Temp_Froid + S_Cmd_Regul_PID_Deshu;
Cons_Actionneur_V3V_Froid_CTA := LIMIT(Cons_Mini_V3V_Bat_Froid, Calcul1, Cons_Maxi_V3V_Bat_Froid);

(**********************************************Décallage de la vitesse du moteur si demande de déshu importante*)
SCL_Real_Decal_Deshu(
	IN_REAL:= S_Cmd_Regul_PID_Deshu,
	LIM_MIN_IN_REAL:= Mini_Decal_PID_Deshu,
	LIM_MAX_IN_REAL:= Maxi_Decal_PID_Deshu,
	LIM_MIN_OUT_REAL:= Mini_Decal_Deshu,
	LIM_MAX_OUT_REAL:= Maxi_Decal_Deshu);
Lect_Cons_VitMot_Cabine_MEnCond := Lect_Cons_VitMot_Cabine_MEnCond;

(**********************************************Gestion du moteur 1 de soufflage de la CTA*)
IF (Dmd_Post_Ventilation OR Mode_Depollution_cycle1)
	THEN
	Cons_Actionneur_Mot1_Souf_CTA := 100.0;
	ELSE
	Cons_Actionneur_Mot1_Souf_CTA := LIMIT(0.0, Lect_Cons_VitMot_Cabine_MEnCond, Cons_Maxi_Mot1_CTA);
END_IF;

(**********************************************Gestion du moteur 2 de soufflage de la CTA*)
IF (Dmd_Post_Ventilation OR Mode_Depollution_cycle1)
	THEN
	Cons_Actionneur_Mot2_Souf_CTA := 100.0;
	ELSE
Cons_Actionneur_Mot2_Souf_CTA := LIMIT(0.0, Lect_Cons_VitMot_Cabine_MEnCond, Cons_Maxi_Mot2_CTA);
END_IF;

(**********************************************Gestion de la batterie electrique*)
(*Consigne ANA*)
Cons_Actionneur_BatElec_CTA := LIMIT(0.0, S_Cmd_Regul_PID_Temp_Chaud, Cons_Maxi_Bat_Electrique);
(*Commande TOR*)
IF (NOT Defaut_Sonde_Temp_Cabine AND NOT Defaut_Alim_BatElec_CTA AND RS_MEnCond.Q1)
THEN Cmd_Actionneur_BatElec_CTA := TRUE;	ELSE Cmd_Actionneur_BatElec_CTA := FALSE;	END_IF;

(**********************************************Gestion de l'humidificateur*)
(*Consigne ANA*)
Cons_Actionneur_Humi_CTA := LIMIT(mini_humi, S_Cmd_Regul_PID_Humi,Cons_Maxi_Humidificateur);

(*Commande TOR*)
IF (RS_MEnCond.Q1 AND NOT Defaut_General_Humi AND E_Pressostat_Secu)
THEN Cmd_Actionneur_Humi_CTA := TRUE;	ELSE Cmd_Actionneur_Humi_CTA := FALSE;	END_IF;

END_PROGRAM

// ---- POUs/Gestion_Enceinte_Clim/F_Gestion_Actionneurs.TcPOU
PROGRAM F_Gestion_Actionneurs
VAR
	V3V_Bat_Froid_CTA		: Servomoteur_V1;
	Batterie_Elec_CTA		: BatElec;
	Humidificateur			: Humidificateur;
	F_Humi: REAL;
	EF_Humi: BOOL;
	F_BatElec: REAL;
	EF_BatElec: BOOL;
END_VAR
VAR // added by the converter: edge detectors and wires of the graphical bodies
    _w1, _w2 : BOOL;
END_VAR

V3V_Bat_Froid_CTA(
    Enable := TRUE,
    Type_Consigne := TRUE,
    Mode_Vidange := FALSE,
    Cons_Pos_Dem := Cons_Actionneur_V3V_Froid_CTA,
    Cmd_Ouv_Dem := FALSE,
    Info_Mes_Pos := 0.0,
    Presence_Fdc := 0,
    Info_Fdc_Ouvert := FALSE,
    Info_Fdc_Ferme := FALSE,
    Secu_Niveau_Haut := FALSE,
    Control_Discrodance := FALSE,
    Hyst_Al_Discord := 0.0,
    Tempo_Discord_TOR := T#0s,
    EF_Forcage := EF_Cons_V3V_Bat_Froid_CTA,
    F_STOR_Registre := FALSE,
    F_SAN_Registre := F_Cons_V3V_Bat_Froid_CTA,
    Defaut_Alim_Eau := FALSE,
    E_Cmd_Rearmement := FALSE,
    In_SCL_In_MIN_REAL := 0.0,
    In_SCL_In_MAX_REAL := 100.0,
    In_SCL_Out_MIN_REAL := 1638.0,
    In_SCL_Out_MAX_REAL := 32767.0); // Servomoteur_V1
S_Cons_V3V_Froid_CTA := V3V_Bat_Froid_CTA.SAN_Cons_Registre;
_w1 := Cons_Actionneur_Mot1_Souf_CTA >= 5.0;
MotRep_CTA(
    Enable := TRUE,
    Cons_Vit_Dem := Cons_Actionneur_Mot1_Souf_CTA,
    Cmd_Ma_Dem := _w1,
    Pres_Mes_Freq := FALSE,
    Info_Freq := Cons_Actionneur_Mot1_Souf_CTA,
    Freq_Min := 0.0,
    Freq_Max := 100.0,
    Info_Marche := _w1,
    Info_Defaut := Defaut_MotRep_CTA,
    ModeOccupe := FALSE,
    Sel_Cons_Fixe := FALSE,
    Inverse_SAN := FALSE,
    SAN_MIN := 0.0,
    SAN_MAX := 32767.0,
    Tab_Var := Tab_MotRep_CTA); // Moteur_EC
S_Cons_MotRep_CTA := MotRep_CTA.SAN_CONS_VAR;
_w2 := Cons_Actionneur_Mot2_Souf_CTA >= 5.0;
MotSouf_CTA(
    Enable := TRUE,
    Cons_Vit_Dem := Cons_Actionneur_Mot2_Souf_CTA,
    Cmd_Ma_Dem := _w2,
    Pres_Mes_Freq := FALSE,
    Info_Freq := Cons_Actionneur_Mot2_Souf_CTA,
    Freq_Min := 0.0,
    Freq_Max := 100.0,
    Info_Marche := _w2,
    Info_Defaut := Defaut_MotSouf_CTA,
    ModeOccupe := FALSE,
    Sel_Cons_Fixe := FALSE,
    Inverse_SAN := FALSE,
    SAN_MIN := 0.0,
    SAN_MAX := 32767.0,
    Tab_Var := Tab_MotSouf_CTA); // Moteur_EC
S_Cons_MotSouf_CTA := MotSouf_CTA.SAN_CONS_VAR;
Batterie_Elec_CTA(
    Enable := TRUE,
    Cons_BatElec_Dem := SEL(EF_BatElec, Cons_Actionneur_BatElec_CTA, F_BatElec),
    Cmd_BatElec_Dem := Cmd_Actionneur_BatElec_CTA,
    Mes_Temp := Tab_MES_Sonde_Temp_Amb.R_MesCor,
    Info_Defaut := NOT Defaut_Alim_BatElec_CTA,
    Info_Ma_Mot := TRUE,
    Info_Press_Sec := E_Pressostat_Secu,
    Type_Commande := TRUE,
    Inverse_SAN := FALSE,
    SAN_MIN := 0.0,
    SAN_MAX := 32767.0,
    Tab_BatElec := Tab_Batterie_Elec_CTA); // BatElec
S_Cons_BatElec_CTA := Batterie_Elec_CTA.SAN_CONS_BAT_ELEC;
S_Cmd_BatElec_CTA := Batterie_Elec_CTA.STOR_CMD_BAT_ELEC;
Humidificateur(
    Enable := TRUE,
    Cmd_Humidificateur := Cmd_Actionneur_Humi_CTA,
    Cons_Humi_Dem := SEL(EF_Humi, Cons_Actionneur_Humi_CTA, F_Humi),
    Info_Defaut := Defaut_Humi_CTA,
    Inverse_SAN := FALSE,
    SAN_OUT_MIN := 0.0,
    SAN_OUT_MAX := 32767.0);
S_Cons_Humi_CTA := Humidificateur.SAN_CONS_HUMI;
S_Cmd_Humi_CTA := Humidificateur.STOR_CMD_HUMI;

END_PROGRAM

